Yaskawa INFORM job: DEMO_NAIHAN_0625_2PAINT_0.JBI

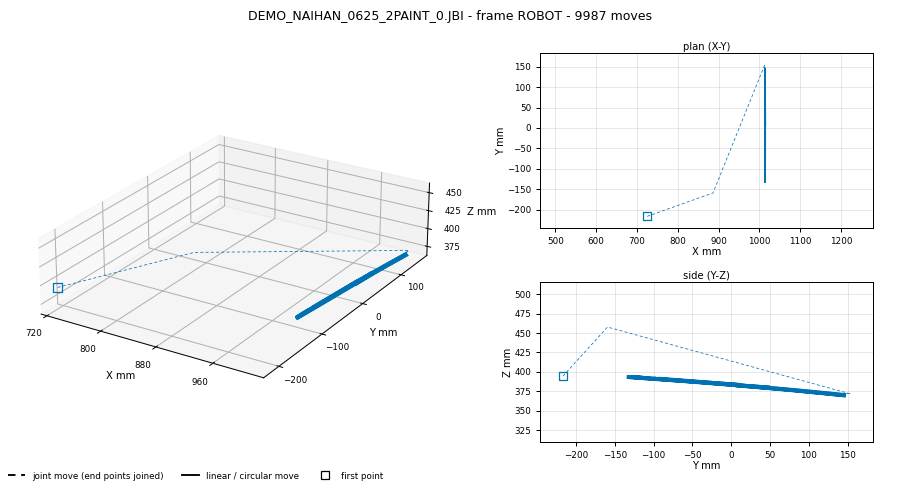
[picture p0: tool path of DEMO_NAIHAN_0625_2PAINT_0.JBI in frame ROBOT, 9987 of 9987 moves have a stored position in this frame; points joined in program order, loops and branches not executed]
/JOB
//NAME DEMO_NAIHAN_0625_2PAINT
//POS
///NPOS 9987,0,0,0,0,0
///TOOL 1
///USER 0
///POSTYPE ROBOT
///RECTAN
///RCONF 1,0,0,0,0,0,0,0,0,0,0,0,0,0,0,0,0,0,0,0,0,0,0,0
C00000=724.889,-216.680,394.500,-180.000,-0.000,-0.000
///USER 0
///POSTYPE ROBOT
///RECTAN
///RCONF 0,0,0,0,0,0,0,0,0,0,0,0,0,0,0,0,0,0,0,0,0,0,0,0
C00001=886.160,-159.406,457.717,-85.028,-4.406,-90.070
///RCONF 1,0,0,0,0,0,0,0,0,0,0,0,0,0,0,0,0,0,0,0,0,0,0,0
C00002=1012.315,153.041,371.808,165.953,61.802,161.272
///RCONF 1,0,0,0,1,0,0,0,0,0,0,0,0,0,0,0,0,0,0,0,0,0,0,0
C00003=1012.444,147.263,372.118,165.953,61.802,161.272
C00004=1012.445,146.855,372.160,165.949,61.816,161.274
C00005=1012.446,146.448,372.202,165.946,61.830,161.276
C00006=1012.447,146.042,372.243,165.944,61.843,161.278
C00007=1012.448,145.637,372.284,165.940,61.857,161.280
C00008=1012.449,145.231,372.325,165.937,61.871,161.282
C00009=1012.450,144.826,372.367,165.934,61.885,161.284
C00010=1012.451,144.422,372.407,165.931,61.898,161.286
C00011=1012.452,144.018,372.449,165.929,61.912,161.288
C00012=1012.453,143.614,372.490,165.925,61.926,161.289
C00013=1012.454,143.211,372.531,165.923,61.939,161.291
C00014=1012.456,142.810,372.572,165.919,61.952,161.293
C00015=1012.456,142.409,372.612,165.917,61.965,161.295
C00016=1012.457,142.007,372.653,165.913,61.979,161.297
C00017=1012.458,141.808,372.673,165.912,61.986,161.298
C00018=1012.459,141.543,372.701,165.910,61.995,161.299
C00019=1012.459,141.136,372.742,165.908,62.008,161.301
C00020=1012.460,140.919,372.763,165.906,62.015,161.302
C00021=1012.461,140.708,372.785,165.904,62.023,161.303
C00022=1012.461,140.481,372.808,165.903,62.030,161.304
C00023=1012.461,140.239,372.832,165.900,62.037,161.305
C00024=1012.462,139.985,372.858,165.899,62.046,161.306
C00025=1012.463,139.724,372.885,165.897,62.054,161.307
C00026=1012.464,139.462,372.911,165.895,62.064,161.309
C00027=1012.464,139.204,372.937,165.894,62.072,161.310
C00028=1012.465,138.956,372.963,165.891,62.080,161.311
C00029=1012.465,138.720,372.986,165.890,62.088,161.312
C00030=1012.466,138.501,373.009,165.889,62.095,161.314
C00031=1012.467,138.104,373.049,165.886,62.107,161.315
C00032=1012.467,137.804,373.079,165.884,62.117,161.316
C00033=1012.469,137.455,373.114,165.882,62.129,161.318
C00034=1012.470,137.112,373.149,165.879,62.140,161.320
C00035=1012.470,136.790,373.181,165.877,62.151,161.321
C00036=1012.471,136.470,373.214,165.875,62.161,161.323
C00037=1012.472,136.129,373.248,165.873,62.172,161.324
C00038=1012.473,135.760,373.285,165.870,62.184,161.326
C00039=1012.474,135.350,373.326,165.867,62.198,161.328
C00040=1012.475,135.091,373.353,165.865,62.207,161.329
C00041=1012.475,134.860,373.376,165.865,62.215,161.331
C00042=1012.476,134.465,373.416,165.862,62.227,161.333
C00043=1012.478,134.070,373.455,165.859,62.240,161.334
C00044=1012.478,133.676,373.495,165.856,62.253,161.336
C00045=1012.479,133.281,373.535,165.854,62.264,161.338
C00046=1012.481,132.887,373.574,165.852,62.276,161.340
C00047=1012.482,132.493,373.615,165.848,62.289,161.341
C00048=1012.482,132.098,373.654,165.846,62.303,161.343
C00049=1012.483,131.704,373.693,165.844,62.316,161.345
C00050=1012.484,131.309,373.733,165.841,62.328,161.347
C00051=1012.486,130.915,373.773,165.839,62.340,161.349
C00052=1012.487,130.520,373.812,165.836,62.353,161.351
C00053=1012.488,130.126,373.852,165.834,62.364,161.352
C00054=1012.489,129.732,373.891,165.831,62.376,161.354
C00055=1012.489,129.338,373.931,165.830,62.388,161.356
C00056=1012.491,128.943,373.970,165.827,62.401,161.358
C00057=1012.492,128.549,374.010,165.824,62.414,161.360
C00058=1012.493,128.154,374.049,165.821,62.426,161.362
C00059=1012.493,127.760,374.089,165.819,62.438,161.363
C00060=1012.495,127.366,374.128,165.816,62.451,161.365
C00061=1012.496,126.972,374.168,165.814,62.463,161.367
C00062=1012.498,126.577,374.207,165.812,62.474,161.368
C00063=1012.498,126.183,374.247,165.810,62.486,161.370
C00064=1012.499,125.789,374.286,165.807,62.498,161.372
C00065=1012.500,125.394,374.325,165.806,62.511,161.374
C00066=1012.501,125.000,374.364,165.803,62.524,161.376
C00067=1012.502,124.605,374.404,165.801,62.535,161.378
C00068=1012.503,124.212,374.444,165.799,62.547,161.380
C00069=1012.504,123.817,374.482,165.796,62.559,161.381
C00070=1012.505,123.422,374.522,165.794,62.571,161.383
C00071=1012.507,123.029,374.561,165.792,62.581,161.385
C00072=1012.507,122.634,374.600,165.790,62.594,161.387
C00073=1012.509,122.240,374.639,165.787,62.606,161.388
C00074=1012.509,121.846,374.679,165.785,62.619,161.391
C00075=1012.511,121.451,374.718,165.783,62.630,161.392
C00076=1012.512,121.057,374.757,165.781,62.642,161.394
C00077=1012.512,120.663,374.797,165.778,62.653,161.395
C00078=1012.514,120.268,374.836,165.776,62.665,161.397
C00079=1012.515,119.874,374.874,165.774,62.675,161.399
C00080=1012.516,119.480,374.914,165.772,62.687,161.401
C00081=1012.517,119.086,374.953,165.769,62.700,161.402
C00082=1012.518,118.692,374.992,165.767,62.712,161.404
C00083=1012.519,118.297,375.031,165.765,62.724,161.406
C00084=1012.520,117.903,375.071,165.764,62.736,161.408
C00085=1012.521,117.509,375.109,165.761,62.747,161.410
C00086=1012.522,117.114,375.149,165.759,62.758,161.411
C00087=1012.524,116.720,375.188,165.757,62.769,161.413
C00088=1012.525,116.326,375.226,165.755,62.780,161.415
C00089=1012.525,115.932,375.266,165.753,62.792,161.417
C00090=1012.526,115.537,375.305,165.750,62.804,161.418
C00091=1012.527,115.143,375.343,165.749,62.816,161.420
C00092=1012.528,114.748,375.383,165.747,62.827,161.422
C00093=1012.529,114.354,375.421,165.745,62.838,161.424
C00094=1012.531,113.960,375.460,165.743,62.849,161.425
C00095=1012.532,113.566,375.499,165.742,62.860,161.427
C00096=1012.532,113.172,375.538,165.739,62.870,161.428
C00097=1012.534,112.777,375.577,165.736,62.882,161.430
C00098=1012.535,112.383,375.616,165.735,62.894,161.432
C00099=1012.536,111.989,375.654,165.732,62.906,161.434
C00100=1012.537,111.594,375.694,165.731,62.917,161.436
C00101=1012.538,111.200,375.732,165.729,62.928,161.437
C00102=1012.539,110.806,375.771,165.726,62.938,161.439
C00103=1012.540,110.412,375.810,165.725,62.949,161.440
C00104=1012.540,110.017,375.849,165.723,62.959,161.442
C00105=1012.542,109.623,375.888,165.722,62.971,161.444
C00106=1012.543,109.229,375.926,165.719,62.982,161.446
C00107=1012.544,108.835,375.965,165.718,62.994,161.448
C00108=1012.545,108.441,376.003,165.715,63.005,161.449
C00109=1012.546,108.045,376.042,165.714,63.016,161.451
C00110=1012.547,107.651,376.081,165.711,63.026,161.452
C00111=1012.548,107.257,376.119,165.710,63.037,161.454
C00112=1012.550,106.863,376.158,165.708,63.047,161.455
C00113=1012.550,106.468,376.197,165.706,63.058,161.457
C00114=1012.551,106.074,376.235,165.704,63.069,161.459
C00115=1012.552,105.680,376.274,165.703,63.080,161.461
C00116=1012.554,105.285,376.313,165.700,63.092,161.463
C00117=1012.555,104.891,376.351,165.698,63.102,161.464
C00118=1012.555,104.496,376.390,165.697,63.113,161.466
C00119=1012.556,104.102,376.428,165.694,63.123,161.467
C00120=1012.557,103.708,376.467,165.693,63.132,161.469
C00121=1012.559,103.314,376.506,165.691,63.142,161.470
C00122=1012.560,102.918,376.544,165.690,63.154,161.472
C00123=1012.561,102.524,376.582,165.688,63.165,161.474
C00124=1012.561,102.130,376.621,165.687,63.176,161.476
C00125=1012.563,101.736,376.659,165.685,63.187,161.478
C00126=1012.563,101.341,376.697,165.683,63.197,161.479
C00127=1012.565,100.946,376.737,165.681,63.207,161.480
C00128=1012.566,100.552,376.774,165.680,63.216,161.482
C00129=1012.567,100.158,376.813,165.678,63.226,161.484
C00130=1012.568,99.764,376.851,165.676,63.237,161.485
C00131=1012.569,99.368,376.889,165.675,63.248,161.487
C00132=1012.569,98.974,376.928,165.673,63.259,161.489
C00133=1012.571,98.580,376.966,165.671,63.269,161.490
C00134=1012.572,98.186,377.004,165.669,63.279,161.492
C00135=1012.573,97.790,377.043,165.667,63.289,161.493
C00136=1012.574,97.396,377.081,165.665,63.298,161.495
C00137=1012.575,97.001,377.119,165.664,63.308,161.496
C00138=1012.576,96.607,377.158,165.662,63.318,161.498
C00139=1012.577,96.212,377.196,165.661,63.329,161.500
C00140=1012.578,95.818,377.234,165.659,63.340,161.502
C00141=1012.579,95.423,377.272,165.657,63.350,161.503
C00142=1012.580,95.029,377.310,165.655,63.360,161.504
C00143=1012.581,94.634,377.349,165.654,63.369,161.506
C00144=1012.582,94.239,377.386,165.652,63.380,161.507
C00145=1012.583,93.845,377.425,165.650,63.388,161.509
C00146=1012.583,93.450,377.463,165.649,63.398,161.510
C00147=1012.585,93.055,377.501,165.648,63.407,161.512
C00148=1012.586,92.660,377.539,165.646,63.418,161.513
C00149=1012.586,92.266,377.577,165.643,63.428,161.515
C00150=1012.588,91.871,377.615,165.643,63.438,161.517
C00151=1012.589,91.476,377.653,165.641,63.448,161.518
C00152=1012.590,91.074,377.692,165.639,63.458,161.520
C00153=1012.590,90.827,377.715,165.639,63.464,161.521
C00154=1012.590,90.548,377.743,165.637,63.470,161.522
C00155=1012.592,90.273,377.769,165.636,63.476,161.523
C00156=1012.592,90.039,377.792,165.635,63.482,161.523
C00157=1012.594,89.643,377.830,165.634,63.491,161.525
C00158=1012.595,89.258,377.867,165.632,63.501,161.527
C00159=1012.596,88.879,377.903,165.630,63.510,161.528
C00160=1012.596,88.505,377.940,165.630,63.519,161.530
C00161=1012.598,88.127,377.975,165.628,63.528,161.531
C00162=1012.598,87.742,378.012,165.625,63.537,161.532
C00163=1012.599,87.348,378.050,165.624,63.547,161.534
C00164=1012.600,86.949,378.088,165.623,63.556,161.535
C00165=1012.601,86.548,378.127,165.622,63.566,161.537
C00166=1012.602,86.146,378.166,165.619,63.575,161.538
C00167=1012.603,85.742,378.204,165.618,63.585,161.540
C00168=1012.604,85.338,378.243,165.617,63.595,161.541
C00169=1012.605,84.933,378.282,165.615,63.605,161.543
C00170=1012.605,84.526,378.321,165.613,63.613,161.544
C00171=1012.607,84.117,378.359,165.612,63.623,161.546
C00172=1012.608,83.707,378.399,165.610,63.633,161.547
C00173=1012.608,83.297,378.438,165.609,63.643,161.549
C00174=1012.610,82.884,378.478,165.608,63.652,161.551
C00175=1012.610,82.472,378.517,165.605,63.662,161.552
C00176=1012.612,82.058,378.556,165.604,63.671,161.553
C00177=1012.613,81.643,378.596,165.603,63.681,161.555
C00178=1012.614,81.249,378.633,165.601,63.690,161.556
C00179=1012.614,80.886,378.668,165.599,63.699,161.558
C00180=1012.616,80.503,378.704,165.599,63.707,161.559
C00181=1012.616,80.090,378.744,165.597,63.716,161.560
C00182=1012.617,79.682,378.782,165.595,63.726,161.562
C00183=1012.618,79.279,378.821,165.594,63.734,161.563
C00184=1012.619,78.885,378.858,165.592,63.743,161.565
C00185=1012.620,78.495,378.896,165.590,63.752,161.566
C00186=1012.621,78.112,378.932,165.589,63.761,161.567
C00187=1012.622,77.730,378.968,165.588,63.769,161.569
C00188=1012.623,77.348,379.004,165.586,63.778,161.570
C00189=1012.623,76.961,379.041,165.585,63.786,161.571
C00190=1012.624,76.567,379.078,165.584,63.795,161.573
C00191=1012.626,76.165,379.116,165.582,63.804,161.574
C00192=1012.626,75.757,379.155,165.580,63.813,161.575
C00193=1012.627,75.342,379.194,165.579,63.823,161.577
C00194=1012.627,75.133,379.214,165.578,63.826,161.578
C00195=1012.628,74.918,379.234,165.577,63.831,161.578
C00196=1012.628,74.691,379.256,165.576,63.836,161.579
C00197=1012.629,74.463,379.277,165.576,63.841,161.580
C00198=1012.629,74.244,379.297,165.575,63.846,161.581
C00199=1012.631,73.829,379.338,165.574,63.855,161.582
C00200=1012.631,73.417,379.376,165.572,63.864,161.583
C00201=1012.632,73.008,379.414,165.570,63.873,161.585
C00202=1012.633,72.599,379.453,165.569,63.881,161.586
C00203=1012.633,72.194,379.492,165.568,63.890,161.587
C00204=1012.635,71.788,379.530,165.566,63.899,161.589
C00205=1012.636,71.383,379.568,165.565,63.907,161.590
C00206=1012.637,70.980,379.606,165.563,63.916,161.592
C00207=1012.637,70.574,379.644,165.562,63.925,161.593
C00208=1012.638,70.170,379.682,165.561,63.933,161.594
C00209=1012.640,69.766,379.720,165.559,63.942,161.596
C00210=1012.640,69.358,379.758,165.558,63.950,161.597
C00211=1012.641,68.942,379.797,165.556,63.959,161.598
C00212=1012.641,68.523,379.836,165.554,63.967,161.599
C00213=1012.643,68.112,379.875,165.553,63.976,161.601
C00214=1012.643,67.711,379.912,165.552,63.985,161.602
C00215=1012.645,67.313,379.950,165.550,63.992,161.603
C00216=1012.645,66.915,379.987,165.550,64.001,161.605
C00217=1012.646,66.551,380.022,165.548,64.008,161.606
C00218=1012.647,66.224,380.052,165.547,64.015,161.607
C00219=1012.647,65.831,380.088,165.545,64.022,161.608
C00220=1012.648,65.623,380.108,165.545,64.027,161.609
C00221=1012.648,65.408,380.128,165.544,64.031,161.609
C00222=1012.649,65.189,380.149,165.544,64.036,161.610
C00223=1012.649,64.966,380.169,165.542,64.040,161.611
C00224=1012.649,64.740,380.191,165.542,64.045,161.612
C00225=1012.651,64.514,380.212,165.540,64.049,161.612
C00226=1012.651,64.295,380.232,165.540,64.053,161.613
C00227=1012.651,63.890,380.269,165.537,64.085,161.619
C00228=1012.650,63.679,380.286,165.536,64.150,161.632
C00229=1012.649,63.443,380.305,165.533,64.223,161.647
C00230=1012.648,63.194,380.324,165.530,64.299,161.663
C00231=1012.647,62.952,380.344,165.527,64.374,161.678
C00232=1012.646,62.733,380.362,165.524,64.440,161.692
C00233=1012.645,62.450,380.384,165.522,64.527,161.710
C00234=1012.644,62.051,380.416,165.518,64.647,161.735
C00235=1012.641,61.654,380.447,165.515,64.765,161.760
C00236=1012.640,61.259,380.479,165.512,64.884,161.785
C00237=1012.639,60.863,380.511,165.509,65.001,161.810
C00238=1012.637,60.466,380.543,165.507,65.118,161.835
C00239=1012.635,60.071,380.574,165.504,65.234,161.859
C00240=1012.634,59.675,380.606,165.502,65.350,161.884
C00241=1012.633,59.278,380.638,165.501,65.464,161.910
C00242=1012.631,58.883,380.669,165.499,65.578,161.934
C00243=1012.630,58.486,380.701,165.498,65.692,161.960
C00244=1012.629,58.090,380.733,165.496,65.805,161.985
C00245=1012.627,57.695,380.765,165.496,65.917,162.010
C00246=1012.626,57.298,380.797,165.495,66.028,162.035
C00247=1012.625,56.902,380.828,165.496,66.139,162.060
C00248=1012.624,56.507,380.860,165.496,66.249,162.085
C00249=1012.623,56.110,380.892,165.496,66.358,162.110
C00250=1012.621,55.714,380.924,165.496,66.467,162.135
C00251=1012.620,55.318,380.955,165.496,66.576,162.160
C00252=1012.619,54.922,380.987,165.497,66.683,162.185
C00253=1012.617,54.527,381.019,165.499,66.791,162.211
C00254=1012.616,54.130,381.051,165.500,66.896,162.235
C00255=1012.615,53.734,381.083,165.501,67.002,162.261
C00256=1012.614,53.339,381.115,165.503,67.108,162.286
C00257=1012.613,52.942,381.146,165.506,67.213,162.311
C00258=1012.611,52.547,381.178,165.508,67.317,162.337
C00259=1012.611,52.151,381.210,165.510,67.419,162.362
C00260=1012.609,51.754,381.242,165.513,67.522,162.387
C00261=1012.608,51.358,381.274,165.516,67.624,162.412
C00262=1012.607,50.963,381.306,165.520,67.726,162.438
C00263=1012.606,50.567,381.338,165.523,67.827,162.463
C00264=1012.605,50.171,381.369,165.528,67.928,162.489
C00265=1012.604,49.775,381.401,165.530,68.028,162.514
C00266=1012.603,49.380,381.433,165.536,68.127,162.540
C00267=1012.602,48.983,381.465,165.539,68.226,162.565
C00268=1012.601,48.588,381.496,165.543,68.324,162.591
C00269=1012.600,48.192,381.528,165.550,68.421,162.617
C00270=1012.599,47.796,381.561,165.554,68.518,162.642
C00271=1012.598,47.400,381.592,165.560,68.615,162.668
C00272=1012.597,47.005,381.624,165.564,68.710,162.693
C00273=1012.597,46.610,381.656,165.571,68.806,162.719
C00274=1012.596,46.214,381.688,165.576,68.901,162.745
C00275=1012.595,45.818,381.719,165.582,68.994,162.771
C00276=1012.594,45.422,381.751,165.588,69.088,162.796
C00277=1012.593,45.026,381.783,165.594,69.181,162.822
C00278=1012.592,44.630,381.816,165.602,69.274,162.848
C00279=1012.592,44.236,381.847,165.608,69.365,162.874
C00280=1012.591,43.839,381.879,165.616,69.457,162.900
C00281=1012.590,43.443,381.911,165.623,69.547,162.926
C00282=1012.589,43.048,381.943,165.630,69.637,162.952
C00283=1012.588,42.653,381.975,165.639,69.727,162.978
C00284=1012.588,42.257,382.007,165.646,69.816,163.004
C00285=1012.587,41.861,382.038,165.655,69.905,163.030
C00286=1012.586,41.466,382.070,165.663,69.993,163.056
C00287=1012.586,41.070,382.103,165.671,70.080,163.082
C00288=1012.585,40.675,382.134,165.680,70.167,163.108
C00289=1012.584,40.280,382.166,165.689,70.253,163.134
C00290=1012.584,39.884,382.199,165.698,70.338,163.160
C00291=1012.583,39.489,382.230,165.708,70.424,163.187
C00292=1012.582,39.093,382.261,165.716,70.508,163.213
C00293=1012.582,38.697,382.294,165.727,70.592,163.240
C00294=1012.581,38.302,382.325,165.737,70.676,163.266
C00295=1012.581,37.906,382.358,165.747,70.758,163.292
C00296=1012.580,37.511,382.390,165.756,70.841,163.318
C00297=1012.579,37.116,382.421,165.767,70.922,163.345
C00298=1012.579,36.720,382.454,165.778,71.004,163.371
C00299=1012.578,36.325,382.486,165.788,71.084,163.397
C00300=1012.578,35.930,382.518,165.799,71.164,163.424
C00301=1012.576,35.534,382.550,165.810,71.243,163.450
C00302=1012.576,35.139,382.581,165.820,71.322,163.476
C00303=1012.576,34.744,382.613,165.832,71.401,163.503
C00304=1012.575,34.348,382.645,165.843,71.478,163.529
C00305=1012.575,33.953,382.677,165.855,71.556,163.556
C00306=1012.574,33.557,382.709,165.867,71.631,163.581
C00307=1012.574,33.162,382.741,165.878,71.707,163.608
C00308=1012.573,32.767,382.772,165.891,71.782,163.634
C00309=1012.573,32.371,382.805,165.903,71.857,163.661
C00310=1012.572,31.976,382.837,165.916,71.931,163.687
C00311=1012.572,31.580,382.869,165.928,72.005,163.713
C00312=1012.571,31.185,382.901,165.940,72.077,163.739
C00313=1012.571,30.790,382.933,165.953,72.149,163.765
C00314=1012.571,30.395,382.964,165.966,72.221,163.792
C00315=1012.570,29.999,382.997,165.978,72.292,163.818
C00316=1012.570,29.604,383.029,165.990,72.362,163.843
C00317=1012.570,29.209,383.061,166.004,72.432,163.870
C00318=1012.569,28.815,383.093,166.017,72.502,163.896
C00319=1012.568,28.420,383.125,166.030,72.569,163.921
C00320=1012.568,28.028,383.157,166.043,72.636,163.947
C00321=1012.568,27.634,383.189,166.058,72.703,163.973
C00322=1012.568,27.241,383.221,166.071,72.769,163.998
C00323=1012.567,26.847,383.253,166.085,72.835,164.024
C00324=1012.566,26.450,383.285,166.097,72.900,164.049
C00325=1012.566,26.053,383.318,166.111,72.965,164.075
C00326=1012.566,25.645,383.350,166.124,73.031,164.100
C00327=1012.608,25.661,383.471,165.674,70.447,163.177
C00328=1012.650,25.676,383.593,165.454,67.873,162.444
C00329=1012.652,26.075,383.563,165.449,67.750,162.412
C00330=1012.653,26.473,383.533,165.445,67.626,162.382
C00331=1012.656,26.869,383.504,165.440,67.503,162.350
C00332=1012.657,27.264,383.475,165.437,67.380,162.320
C00333=1012.659,27.657,383.446,165.433,67.258,162.290
C00334=1012.660,28.050,383.416,165.431,67.135,162.261
C00335=1012.662,28.443,383.386,165.427,67.013,162.231
C00336=1012.664,28.838,383.357,165.425,66.890,162.202
C00337=1012.666,29.233,383.327,165.423,66.766,162.173
C00338=1012.667,29.629,383.298,165.422,66.642,162.144
C00339=1012.669,30.024,383.268,165.421,66.519,162.115
C00340=1012.671,30.420,383.239,165.420,66.395,162.087
C00341=1012.673,30.815,383.210,165.418,66.270,162.058
C00342=1012.675,31.211,383.179,165.419,66.146,162.030
C00343=1012.676,31.606,383.150,165.419,66.022,162.002
C00344=1012.679,32.002,383.120,165.419,65.898,161.974
C00345=1012.680,32.397,383.091,165.420,65.772,161.946
C00346=1012.683,32.793,383.061,165.420,65.648,161.918
C00347=1012.684,33.188,383.031,165.422,65.523,161.891
C00348=1012.686,33.584,383.001,165.423,65.398,161.864
C00349=1012.688,33.980,382.971,165.425,65.272,161.837
C00350=1012.690,34.375,382.942,165.427,65.148,161.810
C00351=1012.692,34.770,382.912,165.430,65.022,161.783
C00352=1012.694,35.167,382.882,165.433,64.896,161.756
C00353=1012.695,35.562,382.852,165.436,64.771,161.730
C00354=1012.698,35.957,382.822,165.439,64.645,161.704
C00355=1012.700,36.353,382.792,165.442,64.520,161.677
C00356=1012.701,36.748,382.762,165.446,64.393,161.651
C00357=1012.703,37.144,382.732,165.450,64.267,161.625
C00358=1012.706,37.540,382.702,165.454,64.141,161.599
C00359=1012.707,37.936,382.672,165.459,64.015,161.574
C00360=1012.710,38.331,382.642,165.465,63.888,161.549
C00361=1012.711,38.726,382.612,165.469,63.762,161.523
C00362=1012.713,39.122,382.581,165.475,63.635,161.498
C00363=1012.716,39.518,382.551,165.481,63.509,161.473
C00364=1012.718,39.913,382.521,165.486,63.382,161.448
C00365=1012.720,40.309,382.491,165.493,63.255,161.423
C00366=1012.722,40.705,382.461,165.500,63.128,161.398
C00367=1012.724,41.100,382.431,165.506,63.002,161.373
C00368=1012.726,41.496,382.400,165.513,62.874,161.349
C00369=1012.728,41.892,382.370,165.520,62.747,161.324
C00370=1012.731,42.287,382.340,165.528,62.620,161.300
C00371=1012.732,42.683,382.309,165.535,62.493,161.276
C00372=1012.735,43.079,382.279,165.544,62.367,161.252
C00373=1012.736,43.475,382.249,165.552,62.238,161.228
C00374=1012.739,43.871,382.218,165.561,62.112,161.204
C00375=1012.741,44.267,382.188,165.569,61.985,161.180
C00376=1012.743,44.662,382.158,165.577,61.857,161.156
C00377=1012.745,45.058,382.127,165.587,61.730,161.133
C00378=1012.748,45.454,382.097,165.596,61.602,161.110
C00379=1012.750,45.850,382.066,165.606,61.475,161.086
C00380=1012.752,46.245,382.035,165.615,61.347,161.063
C00381=1012.754,46.641,382.005,165.626,61.220,161.040
C00382=1012.757,47.038,381.974,165.636,61.092,161.017
C00383=1012.759,47.434,381.944,165.646,60.965,160.994
C00384=1012.761,47.829,381.914,165.657,60.838,160.971
C00385=1012.764,48.225,381.882,165.668,60.711,160.948
C00386=1012.765,48.621,381.851,165.678,60.584,160.925
C00387=1012.768,49.017,381.821,165.691,60.456,160.903
C00388=1012.770,49.413,381.789,165.702,60.329,160.881
C00389=1012.773,49.809,381.759,165.714,60.202,160.858
C00390=1012.773,49.925,381.750,165.718,60.165,160.852
C00391=1012.563,19.548,383.847,166.338,73.918,164.472
C00392=1012.562,19.333,383.865,166.346,73.946,164.485
C00393=1012.562,18.920,383.898,166.359,73.998,164.508
C00394=1012.563,18.696,383.916,166.367,74.026,164.520
C00395=1012.562,18.447,383.937,166.375,74.057,164.534
C00396=1012.562,18.198,383.957,166.384,74.088,164.548
C00397=1012.562,17.950,383.977,166.391,74.118,164.561
C00398=1012.562,17.704,383.997,166.400,74.147,164.575
C00399=1012.562,17.454,384.018,166.408,74.177,164.588
C00400=1012.562,17.207,384.038,166.416,74.205,164.601
C00401=1012.562,16.960,384.058,166.423,74.233,164.613
C00402=1012.562,16.714,384.079,166.432,74.261,164.626
C00403=1012.562,16.464,384.099,166.439,74.288,164.639
C00404=1012.561,16.216,384.119,166.446,74.315,164.651
C00405=1012.561,15.968,384.139,166.455,74.342,164.663
C00406=1012.562,15.722,384.161,166.463,74.368,164.676
C00407=1012.562,15.472,384.181,166.470,74.394,164.688
C00408=1012.561,15.223,384.202,166.477,74.419,164.699
C00409=1012.562,14.975,384.222,166.484,74.444,164.710
C00410=1012.562,14.726,384.243,166.491,74.467,164.722
C00411=1012.562,14.476,384.263,166.496,74.491,164.732
C00412=1012.562,14.227,384.283,166.504,74.514,164.744
C00413=1012.561,13.977,384.304,166.512,74.537,164.755
C00414=1012.561,13.727,384.325,166.518,74.558,164.764
C00415=1012.561,13.478,384.345,166.524,74.580,164.774
C00416=1012.562,13.227,384.366,166.529,74.600,164.784
C00417=1012.562,12.977,384.387,166.536,74.619,164.793
C00418=1012.562,12.727,384.408,166.541,74.640,164.803
C00419=1012.562,12.478,384.429,166.546,74.657,164.810
C00420=1012.562,12.230,384.449,166.551,74.674,164.818
C00421=1012.562,11.984,384.470,166.556,74.691,164.827
C00422=1012.562,11.745,384.490,166.560,74.706,164.833
C00423=1012.562,11.497,384.511,166.566,74.721,164.841
C00424=1012.562,11.251,384.532,166.569,74.734,164.847
C00425=1012.563,11.001,384.552,166.573,74.747,164.853
C00426=1012.562,10.747,384.574,166.576,74.758,164.859
C00427=1012.563,10.497,384.595,166.578,74.769,164.863
C00428=1012.562,10.247,384.616,166.581,74.777,164.867
C00429=1012.563,9.999,384.637,166.584,74.784,164.871
C00430=1012.563,9.750,384.659,166.583,74.790,164.872
C00431=1012.564,9.502,384.680,166.585,74.793,164.875
C00432=1012.564,9.253,384.701,166.584,74.794,164.874
C00433=1012.564,9.005,384.723,166.584,74.792,164.873
C00434=1012.564,8.756,384.744,166.581,74.789,164.871
C00435=1012.564,8.508,384.766,166.578,74.780,164.866
C00436=1012.565,8.257,384.789,166.573,74.768,164.860
C00437=1012.566,8.007,384.811,166.565,74.749,164.849
C00438=1012.566,7.756,384.834,166.555,74.723,164.836
C00439=1012.567,7.505,384.857,166.543,74.684,164.817
C00440=1012.569,7.092,384.899,166.501,74.562,164.756
C00441=1012.572,6.931,384.924,166.429,74.336,164.647
C00442=1012.576,7.213,384.915,166.334,74.017,164.499
C00443=1012.579,7.492,384.899,166.286,73.844,164.421
C00444=1012.579,7.769,384.882,166.248,73.701,164.359
C00445=1012.581,8.044,384.864,166.213,73.571,164.302
C00446=1012.582,8.293,384.849,166.187,73.462,164.256
C00447=1012.584,8.542,384.832,166.159,73.358,164.212
C00448=1012.585,8.790,384.815,166.135,73.258,164.170
C00449=1012.586,9.037,384.799,166.113,73.162,164.131
C00450=1012.587,9.286,384.782,166.092,73.068,164.093
C00451=1012.588,9.536,384.765,166.070,72.975,164.055
C00452=1012.589,9.786,384.747,166.050,72.884,164.019
C00453=1012.591,10.036,384.730,166.032,72.794,163.984
C00454=1012.591,10.286,384.712,166.011,72.706,163.948
C00455=1012.592,10.537,384.695,165.994,72.620,163.916
C00456=1012.593,10.787,384.677,165.976,72.534,163.882
C00457=1012.594,11.035,384.661,165.960,72.449,163.850
C00458=1012.595,11.282,384.643,165.943,72.366,163.819
C00459=1012.596,11.527,384.625,165.928,72.284,163.789
C00460=1012.597,11.773,384.608,165.911,72.202,163.758
C00461=1012.598,12.024,384.590,165.897,72.120,163.728
C00462=1012.599,12.276,384.572,165.882,72.037,163.698
C00463=1012.599,12.531,384.554,165.867,71.954,163.667
C00464=1012.600,12.787,384.535,165.852,71.872,163.638
C00465=1012.602,13.042,384.518,165.839,71.789,163.609
C00466=1012.602,13.291,384.500,165.825,71.709,163.581
C00467=1012.603,13.540,384.482,165.812,71.630,163.553
C00468=1012.604,13.788,384.464,165.801,71.552,163.526
C00469=1012.605,14.037,384.446,165.788,71.472,163.499
C00470=1012.606,14.286,384.428,165.775,71.394,163.472
C00471=1012.607,14.535,384.410,165.765,71.316,163.446
C00472=1012.608,14.784,384.392,165.752,71.237,163.419
C00473=1012.609,15.032,384.375,165.742,71.159,163.393
C00474=1012.609,15.281,384.357,165.731,71.082,163.368
C00475=1012.611,15.530,384.338,165.720,71.003,163.342
C00476=1012.611,15.780,384.320,165.709,70.926,163.317
C00477=1012.612,16.030,384.302,165.698,70.848,163.291
C00478=1012.613,16.279,384.283,165.689,70.771,163.267
C00479=1012.614,16.530,384.266,165.679,70.693,163.242
C00480=1012.616,16.780,384.247,165.670,70.616,163.217
C00481=1012.616,17.032,384.229,165.660,70.538,163.193
C00482=1012.617,17.282,384.211,165.650,70.460,163.168
C00483=1012.618,17.532,384.193,165.643,70.383,163.145
C00484=1012.619,17.784,384.174,165.634,70.305,163.121
C00485=1012.620,18.035,384.157,165.625,70.228,163.097
C00486=1012.621,18.285,384.138,165.616,70.151,163.073
C00487=1012.622,18.536,384.119,165.608,70.074,163.050
C00488=1012.623,18.787,384.101,165.602,69.997,163.027
C00489=1012.624,19.039,384.083,165.593,69.919,163.004
C00490=1012.625,19.445,384.053,165.582,69.794,162.967
C00491=1012.627,19.860,384.022,165.570,69.666,162.930
C00492=1012.628,20.097,384.005,165.563,69.594,162.909
C00493=1012.629,20.355,383.986,165.556,69.515,162.886
C00494=1012.630,20.622,383.966,165.548,69.432,162.862
C00495=1012.631,20.890,383.947,165.543,69.350,162.839
C00496=1012.632,21.151,383.928,165.536,69.270,162.816
C00497=1012.633,21.394,383.910,165.530,69.195,162.795
C00498=1012.634,21.619,383.893,165.525,69.125,162.776
C00499=1012.636,22.009,383.864,165.516,69.005,162.742
C00500=1012.637,22.235,383.847,165.511,68.936,162.723
C00501=1012.637,22.496,383.828,165.505,68.855,162.701
C00502=1012.638,22.731,383.811,165.502,68.783,162.682
C00503=1012.639,22.936,383.796,165.498,68.720,162.665
C00504=1012.640,23.172,383.778,165.492,68.647,162.645
C00505=1012.641,23.403,383.762,165.488,68.576,162.626
C00506=1012.642,23.662,383.742,165.485,68.496,162.605
C00507=1012.643,23.967,383.719,165.479,68.402,162.580
C00508=1012.645,24.277,383.697,165.474,68.306,162.555
C00509=1012.645,24.606,383.672,165.468,68.204,162.528
C00510=1012.647,24.943,383.647,165.463,68.100,162.501
C00511=1012.649,25.279,383.622,165.459,67.996,162.475
C00512=1012.608,25.267,383.502,165.684,70.540,163.205
C00513=1012.566,25.254,383.382,166.140,73.093,164.126
C00514=1012.566,25.655,383.349,166.125,73.029,164.100
C00515=1012.566,25.407,383.369,166.134,73.069,164.116
C00516=1012.566,25.161,383.389,166.142,73.108,164.131
C00517=1012.565,24.749,383.423,166.157,73.173,164.158
C00518=1012.606,24.817,383.537,165.697,70.641,163.237
C00519=1012.566,24.864,383.414,166.152,73.155,164.150
C00520=1012.567,25.258,383.381,166.139,73.092,164.126
C00521=1012.566,25.009,383.401,166.147,73.131,164.141
C00522=1012.565,24.758,383.422,166.156,73.171,164.157
C00523=1012.566,24.509,383.442,166.165,73.210,164.173
C00524=1012.566,24.265,383.462,166.174,73.247,164.188
C00525=1012.565,24.022,383.482,166.183,73.284,164.204
C00526=1012.565,23.799,383.500,166.190,73.318,164.217
C00527=1012.565,23.420,383.531,166.204,73.376,164.242
C00528=1012.565,23.183,383.550,166.211,73.411,164.256
C00529=1012.564,22.945,383.569,166.220,73.446,164.270
C00530=1012.564,22.675,383.592,166.229,73.487,164.287
C00531=1012.564,22.351,383.618,166.241,73.534,164.307
C00532=1012.564,22.116,383.637,166.249,73.567,164.321
C00533=1012.564,21.885,383.656,166.257,73.601,164.335
C00534=1012.564,21.597,383.679,166.268,73.641,164.353
C00535=1012.563,21.269,383.706,166.279,73.687,164.372
C00536=1012.563,21.013,383.727,166.287,73.722,164.387
C00537=1012.563,20.748,383.749,166.297,73.758,164.403
C00538=1012.564,20.478,383.770,166.306,73.795,164.419
C00539=1012.563,20.214,383.792,166.316,73.831,164.435
C00540=1012.563,19.973,383.812,166.323,73.862,164.448
C00541=1012.563,19.751,383.830,166.330,73.892,164.461
C00542=1012.563,19.548,383.847,166.338,73.918,164.472
C00543=1012.629,-93.771,392.738,165.388,72.408,163.533
C00544=1012.625,-93.572,392.712,165.447,72.663,163.632
C00545=1012.618,-93.811,392.708,165.547,73.088,163.799
C00546=1012.618,-94.073,392.721,165.566,73.174,163.833
C00547=1012.616,-94.335,392.737,165.578,73.226,163.853
C00548=1012.616,-94.597,392.752,165.586,73.262,163.867
C00549=1012.640,-94.959,392.854,165.225,71.642,163.251
C00550=1012.643,-95.343,392.888,165.187,71.445,163.182
C00551=1012.645,-95.723,392.922,165.153,71.261,163.119
C00552=1012.648,-96.102,392.956,165.121,71.084,163.059
C00553=1012.615,-96.298,392.863,165.586,73.314,163.882
C00554=1012.651,-96.479,392.988,165.090,70.913,163.001
C00555=1012.649,-96.226,392.966,165.112,71.028,163.040
C00556=1012.647,-95.971,392.944,165.130,71.144,163.078
C00557=1012.646,-95.723,392.922,165.154,71.262,163.120
C00558=1012.643,-95.472,392.900,165.176,71.382,163.161
C00559=1012.642,-95.223,392.877,165.200,71.506,163.204
C00560=1012.641,-94.972,392.854,165.224,71.635,163.249
C00561=1012.638,-94.723,392.832,165.251,71.769,163.297
C00562=1012.636,-94.473,392.809,165.281,71.911,163.349
C00563=1012.634,-94.223,392.784,165.314,72.066,163.406
C00564=1012.631,-93.972,392.759,165.351,72.240,163.470
C00565=1012.629,-93.771,392.738,165.388,72.408,163.533
C00566=1012.844,-122.010,395.059,164.569,61.082,160.666
C00567=1012.842,-121.711,395.036,164.565,61.193,160.686
C00568=1012.838,-121.322,395.007,164.561,61.338,160.712
C00569=1012.835,-120.934,394.976,164.556,61.483,160.738
C00570=1012.831,-120.546,394.946,164.553,61.628,160.765
C00571=1012.828,-120.157,394.916,164.549,61.773,160.792
C00572=1012.824,-119.769,394.885,164.546,61.919,160.819
C00573=1012.821,-119.380,394.855,164.542,62.064,160.845
C00574=1012.817,-118.992,394.825,164.541,62.210,160.873
C00575=1012.814,-118.604,394.794,164.538,62.356,160.900
C00576=1012.811,-118.215,394.764,164.536,62.502,160.928
C00577=1012.808,-117.827,394.734,164.534,62.647,160.956
C00578=1012.805,-117.439,394.703,164.532,62.794,160.984
C00579=1012.801,-117.050,394.672,164.532,62.940,161.012
C00580=1012.798,-116.661,394.642,164.531,63.087,161.041
C00581=1012.795,-116.273,394.612,164.530,63.233,161.069
C00582=1012.791,-115.885,394.580,164.530,63.379,161.098
C00583=1012.788,-115.496,394.550,164.530,63.526,161.127
C00584=1012.785,-115.107,394.519,164.530,63.673,161.157
C00585=1012.782,-114.718,394.488,164.531,63.819,161.186
C00586=1012.779,-114.330,394.457,164.532,63.966,161.216
C00587=1012.776,-113.942,394.426,164.533,64.114,161.246
C00588=1012.772,-113.553,394.395,164.535,64.260,161.276
C00589=1012.770,-113.164,394.364,164.538,64.407,161.307
C00590=1012.767,-112.775,394.333,164.540,64.554,161.338
C00591=1012.764,-112.387,394.302,164.542,64.701,161.369
C00592=1012.760,-111.998,394.271,164.546,64.848,161.400
C00593=1012.757,-111.610,394.240,164.550,64.995,161.432
C00594=1012.755,-111.221,394.208,164.554,65.143,161.464
C00595=1012.752,-110.832,394.178,164.558,65.290,161.496
C00596=1012.749,-110.443,394.146,164.564,65.437,161.528
C00597=1012.746,-110.054,394.115,164.568,65.584,161.561
C00598=1012.743,-109.665,394.083,164.574,65.732,161.594
C00599=1012.740,-109.276,394.052,164.581,65.880,161.627
C00600=1012.737,-108.871,394.019,164.587,66.033,161.662
C00601=1012.735,-108.660,394.001,164.591,66.113,161.681
C00602=1012.734,-108.441,393.985,164.595,66.196,161.700
C00603=1012.732,-108.216,393.966,164.599,66.282,161.720
C00604=1012.731,-107.987,393.947,164.604,66.369,161.740
C00605=1012.729,-107.754,393.929,164.607,66.457,161.760
C00606=1012.727,-107.521,393.910,164.612,66.545,161.781
C00607=1012.725,-107.292,393.891,164.616,66.633,161.802
C00608=1012.723,-107.065,393.872,164.622,66.719,161.822
C00609=1012.722,-106.844,393.855,164.626,66.803,161.843
C00610=1012.719,-106.424,393.820,164.637,66.963,161.881
C00611=1012.717,-106.027,393.788,164.646,67.114,161.918
C00612=1012.714,-105.638,393.756,164.658,67.262,161.955
C00613=1012.671,-105.646,393.637,164.865,69.785,162.620
C00614=1012.629,-105.653,393.519,165.277,72.316,163.451
C00615=1012.630,-106.043,393.547,165.262,72.255,163.427
C00616=1012.631,-106.440,393.575,165.246,72.191,163.402
C00617=1012.632,-106.860,393.606,165.228,72.121,163.374
C00618=1012.633,-107.082,393.622,165.219,72.084,163.360
C00619=1012.633,-107.307,393.638,165.209,72.045,163.345
C00620=1012.633,-107.537,393.654,165.198,72.006,163.330
C00621=1012.634,-107.770,393.671,165.190,71.967,163.315
C00622=1012.635,-108.002,393.688,165.181,71.926,163.300
C00623=1012.636,-108.232,393.704,165.171,71.886,163.285
C00624=1012.637,-108.457,393.720,165.161,71.846,163.269
C00625=1012.637,-108.677,393.736,165.152,71.807,163.255
C00626=1012.638,-109.094,393.766,165.134,71.732,163.227
C00627=1012.639,-109.489,393.795,165.117,71.660,163.200
C00628=1012.640,-109.877,393.822,165.101,71.587,163.173
C00629=1012.641,-110.266,393.851,165.084,71.514,163.146
C00630=1012.643,-110.656,393.879,165.069,71.440,163.120
C00631=1012.643,-111.045,393.907,165.053,71.365,163.093
C00632=1012.644,-111.433,393.935,165.036,71.289,163.066
C00633=1012.646,-111.822,393.964,165.020,71.212,163.039
C00634=1012.647,-112.211,393.991,165.004,71.134,163.011
C00635=1012.648,-112.600,394.019,164.987,71.054,162.983
C00636=1012.649,-112.989,394.048,164.972,70.975,162.956
C00637=1012.651,-113.378,394.075,164.957,70.894,162.929
C00638=1012.652,-113.767,394.103,164.941,70.812,162.901
C00639=1012.653,-114.155,394.131,164.925,70.729,162.873
C00640=1012.655,-114.544,394.160,164.908,70.645,162.845
C00641=1012.656,-114.933,394.188,164.893,70.561,162.817
C00642=1012.657,-115.321,394.217,164.879,70.475,162.790
C00643=1012.659,-115.710,394.244,164.864,70.389,162.762
C00644=1012.661,-116.099,394.273,164.849,70.301,162.733
C00645=1012.662,-116.487,394.300,164.833,70.213,162.705
C00646=1012.663,-116.876,394.329,164.819,70.124,162.677
C00647=1012.664,-117.264,394.357,164.804,70.035,162.649
C00648=1012.666,-117.653,394.385,164.789,69.944,162.620
C00649=1012.668,-118.041,394.414,164.775,69.852,162.592
C00650=1012.669,-118.430,394.442,164.761,69.759,162.563
C00651=1012.671,-118.818,394.470,164.746,69.665,162.535
C00652=1012.673,-119.207,394.499,164.733,69.570,162.506
C00653=1012.674,-119.595,394.527,164.719,69.475,162.478
C00654=1012.675,-119.984,394.555,164.707,69.379,162.450
C00655=1012.677,-120.372,394.584,164.693,69.281,162.421
C00656=1012.678,-120.761,394.612,164.680,69.183,162.393
C00657=1012.680,-121.149,394.640,164.667,69.083,162.364
C00658=1012.682,-121.537,394.669,164.654,68.983,162.335
C00659=1012.684,-121.926,394.697,164.641,68.882,162.306
C00660=1012.686,-122.315,394.726,164.629,68.781,162.278
C00661=1012.687,-122.703,394.754,164.617,68.677,162.249
C00662=1012.690,-123.091,394.782,164.605,68.573,162.220
C00663=1012.691,-123.479,394.810,164.593,68.468,162.192
C00664=1012.693,-123.868,394.839,164.581,68.363,162.163
C00665=1012.695,-124.256,394.867,164.570,68.256,162.134
C00666=1012.697,-124.645,394.896,164.559,68.148,162.106
C00667=1012.700,-125.033,394.924,164.548,68.039,162.077
C00668=1012.701,-125.421,394.952,164.537,67.929,162.047
C00669=1012.704,-125.809,394.980,164.527,67.818,162.019
C00670=1012.706,-126.198,395.009,164.517,67.706,161.990
C00671=1012.708,-126.586,395.037,164.507,67.595,161.961
C00672=1012.709,-126.974,395.066,164.497,67.481,161.932
C00673=1012.712,-127.362,395.094,164.487,67.366,161.904
C00674=1012.714,-127.750,395.123,164.479,67.250,161.875
C00675=1012.716,-128.138,395.151,164.470,67.133,161.846
C00676=1012.718,-128.527,395.180,164.460,67.015,161.817
C00677=1012.721,-128.915,395.208,164.453,66.896,161.789
C00678=1012.723,-129.302,395.237,164.444,66.775,161.759
C00679=1012.725,-129.691,395.266,164.436,66.655,161.730
C00680=1012.727,-130.079,395.294,164.428,66.532,161.701
C00681=1012.730,-130.467,395.323,164.421,66.409,161.672
C00682=1012.733,-130.855,395.351,164.414,66.285,161.644
C00683=1012.735,-131.244,395.380,164.407,66.159,161.615
C00684=1012.737,-131.634,395.409,164.401,66.031,161.586
C00685=1012.740,-132.020,395.438,164.395,65.904,161.557
C00686=1012.743,-132.407,395.466,164.388,65.775,161.527
C00687=1012.746,-132.796,395.495,164.383,65.644,161.498
C00688=1012.748,-133.183,395.524,164.378,65.513,161.469
C00689=1012.751,-133.572,395.553,164.372,65.380,161.440
C00690=1012.753,-133.960,395.581,164.367,65.246,161.411
C00691=1012.820,13.706,384.977,165.533,60.683,160.899
C00692=1012.819,13.328,385.007,165.526,60.761,160.913
C00693=1012.817,12.944,385.036,165.519,60.839,160.927
C00694=1012.816,12.559,385.066,165.511,60.918,160.940
C00695=1012.814,12.177,385.096,165.504,60.995,160.954
C00696=1012.813,11.805,385.125,165.497,61.071,160.967
C00697=1012.812,11.441,385.153,165.491,61.144,160.980
C00698=1012.810,11.076,385.182,165.485,61.216,160.993
C00699=1012.809,10.702,385.210,165.478,61.290,161.006
C00700=1012.808,10.324,385.239,165.472,61.365,161.019
C00701=1012.806,9.948,385.269,165.465,61.438,161.032
C00702=1012.805,9.573,385.299,165.460,61.511,161.045
C00703=1012.804,9.199,385.327,165.454,61.583,161.058
C00704=1012.802,8.825,385.356,165.447,61.655,161.070
C00705=1012.802,8.451,385.385,165.441,61.727,161.083
C00706=1012.800,8.075,385.414,165.435,61.798,161.096
C00707=1012.799,7.697,385.443,165.430,61.868,161.109
C00708=1012.797,7.315,385.474,165.423,61.940,161.121
C00709=1012.796,6.929,385.503,165.418,62.012,161.135
C00710=1012.795,6.538,385.533,165.413,62.083,161.148
C00711=1012.794,6.145,385.564,165.407,62.156,161.161
C00712=1012.793,5.752,385.594,165.402,62.227,161.174
C00713=1012.791,5.362,385.624,165.396,62.298,161.186
C00714=1012.790,4.973,385.655,165.391,62.367,161.199
C00715=1012.788,4.583,385.685,165.386,62.437,161.212
C00716=1012.788,4.192,385.715,165.381,62.505,161.224
C00717=1012.787,3.820,385.744,165.376,62.571,161.236
C00718=1012.785,3.475,385.771,165.372,62.631,161.248
C00719=1012.784,3.152,385.796,165.367,62.687,161.257
C00720=1012.783,2.828,385.821,165.364,62.742,161.268
C00721=1012.783,2.486,385.848,165.359,62.800,161.278
C00722=1012.781,2.115,385.876,165.356,62.863,161.290
C00723=1012.780,1.723,385.907,165.351,62.929,161.302
C00724=1012.779,1.325,385.937,165.347,62.996,161.315
C00725=1012.778,0.928,385.968,165.342,63.061,161.327
C00726=1012.777,0.534,385.999,165.338,63.125,161.339
C00727=1012.776,0.139,386.029,165.333,63.190,161.351
C00728=1012.775,-0.259,386.060,165.329,63.254,161.363
C00729=1012.774,-0.659,386.091,165.326,63.318,161.375
C00730=1012.773,-1.062,386.122,165.321,63.382,161.387
C00731=1012.772,-1.467,386.153,165.317,63.445,161.399
C00732=1012.771,-1.873,386.184,165.313,63.508,161.411
C00733=1012.770,-2.282,386.216,165.309,63.572,161.423
C00734=1012.769,-2.693,386.248,165.305,63.634,161.435
C00735=1012.768,-3.104,386.280,165.302,63.696,161.447
C00736=1012.766,-3.506,386.310,165.299,63.757,161.459
C00737=1012.765,-3.892,386.341,165.295,63.813,161.469
C00738=1012.765,-4.271,386.370,165.292,63.869,161.480
C00739=1012.764,-4.662,386.401,165.288,63.926,161.491
C00740=1012.763,-5.077,386.433,165.284,63.986,161.502
C00741=1012.762,-5.291,386.449,165.283,64.016,161.508
C00742=1012.762,-5.507,386.466,165.281,64.047,161.514
C00743=1012.761,-5.724,386.483,165.280,64.077,161.520
C00744=1012.761,-5.941,386.499,165.278,64.108,161.526
C00745=1012.760,-6.158,386.516,165.277,64.139,161.532
C00746=1012.760,-6.375,386.533,165.275,64.169,161.538
C00747=1012.760,-6.590,386.550,165.273,64.198,161.543
C00748=1012.759,-6.807,386.566,165.271,64.228,161.549
C00749=1012.758,-7.022,386.582,165.271,64.257,161.555
C00750=1012.758,-7.236,386.599,165.268,64.286,161.560
C00751=1012.757,-7.449,386.616,165.267,64.315,161.566
C00752=1012.757,-7.663,386.632,165.265,64.343,161.571
C00753=1012.757,-7.875,386.649,165.264,64.372,161.577
C00754=1012.756,-8.088,386.665,165.262,64.400,161.583
C00755=1012.756,-8.298,386.682,165.260,64.428,161.588
C00756=1012.755,-8.510,386.698,165.259,64.455,161.593
C00757=1012.755,-8.721,386.714,165.258,64.483,161.599
C00758=1012.755,-8.932,386.730,165.256,64.511,161.604
C00759=1012.754,-9.143,386.747,165.255,64.538,161.609
C00760=1012.753,-9.565,386.779,165.252,64.592,161.620
C00761=1012.752,-9.987,386.812,165.250,64.644,161.630
C00762=1012.752,-10.407,386.844,165.248,64.697,161.641
C00763=1012.751,-10.826,386.877,165.243,64.748,161.650
C00764=1012.750,-11.244,386.909,165.242,64.798,161.661
C00765=1012.749,-11.660,386.941,165.239,64.849,161.670
C00766=1012.749,-12.075,386.974,165.237,64.897,161.680
C00767=1012.748,-12.489,387.005,165.235,64.945,161.690
C00768=1012.747,-12.897,387.037,165.232,64.993,161.699
C00769=1012.746,-13.296,387.068,165.230,65.038,161.708
C00770=1012.745,-13.683,387.098,165.228,65.081,161.717
C00771=1012.745,-14.062,387.127,165.227,65.123,161.725
C00772=1012.745,-14.436,387.156,165.224,65.163,161.733
C00773=1012.744,-14.812,387.184,165.222,65.204,161.741
C00774=1012.743,-15.196,387.215,165.220,65.245,161.749
C00775=1012.743,-15.588,387.245,165.218,65.285,161.757
C00776=1012.742,-15.984,387.276,165.217,65.326,161.765
C00777=1012.741,-16.380,387.306,165.213,65.366,161.773
C00778=1012.741,-16.778,387.337,165.212,65.406,161.781
C00779=1012.741,-17.174,387.367,165.210,65.445,161.789
C00780=1012.740,-17.560,387.397,165.208,65.482,161.796
C00781=1012.739,-17.763,387.413,165.207,65.502,161.800
C00782=1012.739,-17.990,387.430,165.207,65.523,161.805
C00783=1012.739,-18.242,387.450,165.205,65.547,161.809
C00784=1012.739,-18.515,387.471,165.204,65.572,161.814
C00785=1012.738,-18.795,387.492,165.202,65.598,161.819
C00786=1012.738,-19.069,387.513,165.200,65.623,161.824
C00787=1012.738,-19.325,387.534,165.200,65.645,161.829
C00788=1012.737,-19.556,387.551,165.199,65.666,161.833
C00789=1012.737,-19.761,387.567,165.198,65.684,161.836
C00790=1012.737,-20.112,387.595,165.196,65.715,161.842
C00791=1012.736,-20.509,387.625,165.195,65.748,161.849
C00792=1012.736,-20.902,387.655,165.193,65.781,161.856
C00793=1012.735,-21.296,387.686,165.192,65.813,161.862
C00794=1012.735,-21.689,387.716,165.189,65.845,161.868
C00795=1012.734,-22.083,387.747,165.188,65.876,161.875
C00796=1012.734,-22.476,387.777,165.186,65.907,161.881
C00797=1012.734,-22.869,387.807,165.185,65.936,161.887
C00798=1012.733,-23.263,387.838,165.183,65.965,161.892
C00799=1012.733,-23.656,387.868,165.181,65.994,161.898
C00800=1012.732,-24.050,387.899,165.180,66.022,161.903
C00801=1012.732,-24.443,387.929,165.178,66.049,161.909
C00802=1012.732,-24.836,387.959,165.176,66.076,161.914
C00803=1012.731,-25.230,387.990,165.174,66.102,161.919
C00804=1012.731,-25.623,388.020,165.172,66.127,161.924
C00805=1012.730,-26.017,388.051,165.171,66.152,161.929
C00806=1012.730,-26.410,388.081,165.169,66.177,161.933
C00807=1012.730,-26.803,388.111,165.167,66.199,161.938
C00808=1012.729,-27.197,388.142,165.165,66.222,161.942
C00809=1012.729,-27.590,388.172,165.165,66.245,161.947
C00810=1012.729,-27.984,388.203,165.163,66.266,161.951
C00811=1012.729,-28.378,388.233,165.160,66.287,161.954
C00812=1012.728,-28.772,388.263,165.159,66.307,161.958
C00813=1012.728,-29.165,388.294,165.157,66.328,161.962
C00814=1012.728,-29.558,388.324,165.156,66.347,161.966
C00815=1012.728,-29.952,388.355,165.154,66.365,161.969
C00816=1012.728,-30.346,388.385,165.152,66.383,161.972
C00817=1012.727,-30.739,388.416,165.151,66.400,161.975
C00818=1012.727,-31.133,388.445,165.149,66.416,161.978
C00819=1012.727,-31.527,388.477,165.147,66.432,161.981
C00820=1012.727,-31.920,388.507,165.144,66.447,161.983
C00821=1012.727,-32.314,388.537,165.143,66.462,161.986
C00822=1012.726,-32.707,388.568,165.140,66.476,161.988
C00823=1012.727,-33.101,388.599,165.139,66.489,161.990
C00824=1012.726,-33.495,388.628,165.137,66.502,161.992
C00825=1012.726,-33.889,388.659,165.136,66.514,161.994
C00826=1012.727,-34.282,388.690,165.133,66.525,161.996
C00827=1012.726,-34.676,388.720,165.131,66.536,161.997
C00828=1012.726,-35.069,388.750,165.129,66.545,161.998
C00829=1012.726,-35.463,388.780,165.126,66.555,162.000
C00830=1012.726,-35.857,388.811,165.124,66.563,162.001
C00831=1012.726,-36.250,388.841,165.122,66.572,162.002
C00832=1012.726,-36.643,388.872,165.120,66.579,162.002
C00833=1012.726,-37.037,388.903,165.118,66.586,162.003
C00834=1012.725,-37.430,388.933,165.117,66.592,162.004
C00835=1012.726,-37.825,388.963,165.114,66.597,162.004
C00836=1012.725,-38.218,388.994,165.111,66.602,162.004
C00837=1012.725,-38.611,389.024,165.110,66.606,162.004
C00838=1012.726,-39.005,389.055,165.108,66.609,162.004
C00839=1012.726,-39.398,389.085,165.106,66.612,162.004
C00840=1012.726,-39.791,389.115,165.103,66.614,162.003
C00841=1012.726,-40.185,389.146,165.101,66.615,162.002
C00842=1012.725,-40.579,389.177,165.099,66.616,162.002
C00843=1012.725,-40.972,389.207,165.096,66.616,162.001
C00844=1012.726,-41.366,389.237,165.093,66.615,161.999
C00845=1012.726,-41.759,389.267,165.091,66.614,161.998
C00846=1012.727,-42.152,389.298,165.089,66.612,161.997
C00847=1012.726,-42.545,389.328,165.086,66.610,161.995
C00848=1012.726,-42.939,389.359,165.083,66.606,161.993
C00849=1012.727,-43.332,389.390,165.082,66.602,161.991
C00850=1012.727,-43.725,389.420,165.078,66.598,161.989
C00851=1012.726,-44.118,389.450,165.076,66.592,161.987
C00852=1012.728,-44.511,389.481,165.074,66.586,161.984
C00853=1012.727,-44.904,389.511,165.071,66.580,161.982
C00854=1012.727,-45.297,389.541,165.069,66.572,161.979
C00855=1012.728,-45.690,389.573,165.065,66.564,161.976
C00856=1012.728,-46.083,389.602,165.063,66.555,161.973
C00857=1012.728,-46.476,389.633,165.060,66.546,161.970
C00858=1012.728,-46.869,389.664,165.056,66.536,161.966
C00859=1012.728,-47.262,389.694,165.053,66.525,161.962
C00860=1012.729,-47.655,389.724,165.051,66.514,161.959
C00861=1012.729,-48.048,389.754,165.049,66.502,161.955
C00862=1012.730,-48.441,389.784,165.045,66.489,161.951
C00863=1012.730,-48.833,389.816,165.042,66.475,161.947
C00864=1012.730,-49.226,389.846,165.040,66.461,161.943
C00865=1012.730,-49.619,389.876,165.036,66.446,161.937
C00866=1012.731,-50.012,389.906,165.034,66.431,161.934
C00867=1012.731,-50.405,389.937,165.030,66.415,161.928
C00868=1012.731,-50.797,389.967,165.028,66.397,161.923
C00869=1012.732,-51.190,389.998,165.024,66.380,161.918
C00870=1012.732,-51.583,390.028,165.021,66.362,161.913
C00871=1012.733,-51.976,390.059,165.018,66.343,161.907
C00872=1012.733,-52.368,390.089,165.015,66.323,161.902
C00873=1012.733,-52.761,390.120,165.013,66.303,161.896
C00874=1012.734,-53.154,390.150,165.009,66.281,161.890
C00875=1012.735,-53.546,390.180,165.005,66.260,161.884
C00876=1012.735,-53.940,390.211,165.003,66.238,161.878
C00877=1012.735,-54.331,390.241,165.000,66.214,161.872
C00878=1012.737,-54.724,390.272,164.996,66.191,161.865
C00879=1012.736,-55.117,390.302,164.994,66.166,161.859
C00880=1012.737,-55.510,390.332,164.991,66.141,161.852
C00881=1012.737,-55.903,390.363,164.987,66.115,161.844
C00882=1012.739,-56.296,390.393,164.984,66.088,161.837
C00883=1012.738,-56.689,390.424,164.980,66.061,161.830
C00884=1012.739,-57.082,390.454,164.978,66.033,161.823
C00885=1012.740,-57.476,390.485,164.974,66.004,161.815
C00886=1012.740,-57.871,390.516,164.971,65.974,161.807
C00887=1012.741,-58.266,390.546,164.968,65.944,161.799
C00888=1012.741,-58.661,390.577,164.964,65.913,161.791
C00889=1012.742,-59.058,390.607,164.961,65.880,161.783
C00890=1012.743,-59.454,390.638,164.957,65.848,161.774
C00891=1012.744,-59.850,390.669,164.954,65.815,161.766
C00892=1012.744,-60.248,390.700,164.951,65.781,161.757
C00893=1012.745,-60.646,390.731,164.947,65.746,161.748
C00894=1012.746,-61.045,390.762,164.945,65.711,161.740
C00895=1012.747,-61.443,390.793,164.941,65.674,161.730
C00896=1012.747,-61.843,390.824,164.938,65.637,161.721
C00897=1012.748,-62.243,390.854,164.935,65.599,161.712
C00898=1012.749,-62.643,390.886,164.931,65.560,161.702
C00899=1012.749,-63.045,390.916,164.928,65.521,161.692
C00900=1012.751,-63.446,390.947,164.925,65.480,161.682
C00901=1012.751,-63.848,390.979,164.921,65.439,161.672
C00902=1012.752,-64.250,391.010,164.918,65.397,161.662
C00903=1012.753,-64.652,391.042,164.915,65.355,161.651
C00904=1012.753,-65.056,391.073,164.912,65.311,161.641
C00905=1012.755,-65.458,391.104,164.910,65.267,161.631
C00906=1012.756,-65.861,391.135,164.906,65.222,161.620
C00907=1012.756,-66.266,391.167,164.903,65.176,161.609
C00908=1012.758,-66.670,391.198,164.900,65.129,161.597
C00909=1012.758,-67.074,391.229,164.897,65.082,161.586
C00910=1012.760,-67.477,391.261,164.894,65.034,161.575
C00911=1012.760,-67.882,391.292,164.891,64.986,161.564
C00912=1012.761,-68.287,391.323,164.888,64.936,161.552
C00913=1012.763,-68.690,391.355,164.885,64.886,161.540
C00914=1012.763,-69.095,391.386,164.882,64.834,161.528
C00915=1012.765,-69.500,391.418,164.879,64.783,161.516
C00916=1012.766,-69.904,391.449,164.877,64.730,161.504
C00917=1012.767,-70.309,391.480,164.874,64.677,161.492
C00918=1012.768,-70.713,391.511,164.871,64.623,161.479
C00919=1012.769,-71.118,391.543,164.869,64.568,161.467
C00920=1012.770,-71.522,391.574,164.865,64.513,161.454
C00921=1012.771,-71.926,391.606,164.862,64.456,161.441
C00922=1012.773,-72.330,391.637,164.860,64.399,161.429
C00923=1012.774,-72.734,391.669,164.858,64.341,161.416
C00924=1012.776,-73.138,391.699,164.855,64.283,161.403
C00925=1012.777,-73.541,391.731,164.853,64.224,161.390
C00926=1012.778,-73.945,391.762,164.851,64.164,161.376
C00927=1012.778,-74.348,391.793,164.849,64.103,161.363
C00928=1012.780,-74.751,391.825,164.847,64.042,161.349
C00929=1012.781,-75.155,391.856,164.845,63.979,161.336
C00930=1012.783,-75.557,391.887,164.842,63.916,161.322
C00931=1012.784,-75.961,391.919,164.841,63.853,161.308
C00932=1012.786,-76.364,391.950,164.839,63.789,161.294
C00933=1012.787,-76.766,391.981,164.836,63.724,161.280
C00934=1012.788,-77.168,392.012,164.835,63.658,161.266
C00935=1012.789,-77.569,392.043,164.834,63.592,161.252
C00936=1012.791,-77.972,392.074,164.832,63.525,161.238
C00937=1012.793,-78.373,392.105,164.830,63.456,161.223
C00938=1012.794,-78.774,392.137,164.828,63.388,161.209
C00939=1012.796,-79.174,392.167,164.827,63.319,161.194
C00940=1012.797,-79.574,392.199,164.827,63.249,161.180
C00941=1012.798,-79.974,392.230,164.826,63.179,161.165
C00942=1012.800,-80.373,392.261,164.824,63.108,161.151
C00943=1012.801,-80.771,392.292,164.823,63.037,161.136
C00944=1012.803,-81.168,392.322,164.822,62.965,161.121
C00945=1012.804,-81.566,392.353,164.821,62.892,161.106
C00946=1012.806,-81.964,392.384,164.821,62.818,161.091
C00947=1012.808,-82.363,392.415,164.820,62.743,161.076
C00948=1012.810,-82.759,392.446,164.820,62.669,161.061
C00949=1012.811,-83.156,392.477,164.819,62.593,161.045
C00950=1012.813,-83.552,392.507,164.819,62.517,161.030
C00951=1012.815,-83.944,392.537,164.818,62.441,161.015
C00952=1012.816,-84.336,392.567,164.818,62.364,160.999
C00953=1012.818,-84.754,392.600,164.818,62.282,160.983
C00954=1012.819,-84.985,392.618,164.818,62.236,160.974
C00955=1012.820,-85.222,392.637,164.819,62.188,160.965
C00956=1012.821,-85.462,392.655,164.819,62.140,160.955
C00957=1012.822,-85.697,392.673,164.820,62.093,160.946
C00958=1012.823,-85.919,392.690,164.819,62.047,160.937
C00959=1012.825,-86.327,392.721,164.820,61.964,160.921
C00960=1012.827,-86.715,392.752,164.821,61.883,160.905
C00961=1012.829,-87.093,392.781,164.821,61.805,160.890
C00962=1012.831,-87.460,392.809,164.821,61.728,160.875
C00963=1012.833,-87.823,392.838,164.824,61.652,160.860
C00964=1012.834,-88.200,392.867,164.824,61.572,160.845
C00965=1012.836,-88.585,392.896,164.825,61.489,160.829
C00966=1012.837,-88.804,392.913,164.826,61.441,160.820
C00967=1012.838,-89.046,392.932,164.827,61.389,160.810
C00968=1012.840,-89.302,392.952,164.828,61.333,160.800
C00969=1012.841,-89.561,392.972,164.828,61.277,160.789
C00970=1012.842,-89.812,392.991,164.829,61.221,160.778
C00971=1012.843,-90.071,393.011,164.831,61.164,160.768
C00972=1012.610,-133.983,395.183,165.422,73.776,163.914
C00973=1012.608,-133.594,395.153,165.467,73.917,163.978
C00974=1012.606,-133.207,395.124,165.512,74.058,164.042
C00975=1012.604,-132.819,395.095,165.558,74.198,164.107
C00976=1012.602,-132.431,395.065,165.605,74.336,164.172
C00977=1012.601,-132.043,395.036,165.654,74.474,164.239
C00978=1012.599,-131.655,395.007,165.703,74.612,164.306
C00979=1012.597,-131.267,394.977,165.754,74.749,164.375
C00980=1012.595,-130.879,394.948,165.807,74.885,164.445
C00981=1012.593,-130.491,394.919,165.860,75.021,164.515
C00982=1012.592,-130.103,394.889,165.913,75.156,164.585
C00983=1012.590,-129.715,394.860,165.968,75.291,164.657
C00984=1012.588,-129.327,394.830,166.024,75.424,164.730
C00985=1012.587,-128.939,394.801,166.082,75.558,164.804
C00986=1012.585,-128.551,394.772,166.141,75.690,164.880
C00987=1012.583,-128.163,394.742,166.201,75.822,164.955
C00988=1012.582,-127.775,394.713,166.262,75.954,165.033
C00989=1012.580,-127.387,394.684,166.324,76.085,165.110
C00990=1012.579,-126.999,394.654,166.386,76.214,165.189
C00991=1012.578,-126.610,394.624,166.452,76.344,165.270
C00992=1012.577,-126.222,394.595,166.517,76.473,165.351
C00993=1012.574,-125.834,394.565,166.585,76.601,165.434
C00994=1012.573,-125.446,394.536,166.653,76.729,165.518
C00995=1012.571,-125.058,394.506,166.725,76.856,165.604
C00996=1012.570,-124.669,394.477,166.797,76.983,165.690
C00997=1012.569,-124.281,394.448,166.869,77.109,165.777
C00998=1012.568,-123.893,394.418,166.944,77.234,165.867
C00999=1012.566,-123.505,394.389,167.020,77.359,165.957
C01000=1012.564,-123.116,394.359,167.098,77.484,166.049
C01001=1012.563,-122.728,394.330,167.177,77.607,166.142
C01002=1012.561,-122.340,394.300,167.259,77.730,166.238
C01003=1012.561,-121.952,394.270,167.341,77.853,166.334
C01004=1012.559,-121.564,394.241,167.426,77.975,166.432
C01005=1012.559,-121.176,394.211,167.512,78.097,166.532
C01006=1012.557,-120.787,394.182,167.598,78.217,166.632
C01007=1012.556,-120.399,394.152,167.688,78.337,166.734
C01008=1012.555,-120.011,394.123,167.778,78.457,166.838
C01009=1012.554,-119.622,394.093,167.871,78.576,166.944
C01010=1012.552,-119.234,394.064,167.968,78.695,167.053
C01011=1012.551,-118.845,394.035,168.065,78.813,167.162
C01012=1012.550,-118.457,394.004,168.162,78.931,167.273
C01013=1012.549,-118.069,393.974,168.264,79.047,167.386
C01014=1012.548,-117.680,393.945,168.366,79.163,167.501
C01015=1012.547,-117.291,393.915,168.471,79.279,167.618
C01016=1012.545,-116.903,393.886,168.580,79.395,167.739
C01017=1012.545,-116.515,393.856,168.690,79.509,167.860
C01018=1012.544,-116.126,393.827,168.800,79.623,167.982
C01019=1012.543,-115.737,393.797,168.914,79.737,168.108
C01020=1012.542,-115.349,393.768,169.029,79.849,168.235
C01021=1012.541,-114.961,393.738,169.148,79.962,168.365
C01022=1012.540,-114.573,393.708,169.271,80.074,168.499
C01023=1012.539,-114.184,393.678,169.393,80.186,168.633
C01024=1012.538,-113.795,393.649,169.519,80.295,168.770
C01025=1012.537,-113.406,393.619,169.647,80.406,168.909
C01026=1012.536,-113.018,393.590,169.780,80.516,169.052
C01027=1012.535,-112.629,393.560,169.915,80.624,169.197
C01028=1012.535,-112.240,393.530,170.052,80.733,169.346
C01029=1012.534,-111.851,393.501,170.192,80.841,169.496
C01030=1012.533,-111.463,393.471,170.337,80.948,169.651
C01031=1012.532,-111.073,393.441,170.481,81.054,169.806
C01032=1012.531,-110.685,393.410,170.631,81.161,169.966
C01033=1012.530,-110.296,393.381,170.782,81.266,170.127
C01034=1012.529,-109.908,393.351,170.938,81.371,170.293
C01035=1012.529,-109.519,393.321,171.100,81.476,170.464
C01036=1012.528,-109.124,393.291,171.264,81.581,170.639
C01037=1012.527,-108.707,393.260,171.445,81.691,170.829
C01038=1012.527,-108.488,393.242,171.540,81.750,170.930
C01039=1012.527,-108.263,393.225,171.636,81.808,171.032
C01040=1012.526,-108.032,393.207,171.741,81.868,171.142
C01041=1012.525,-107.801,393.190,171.847,81.929,171.253
C01042=1012.525,-107.568,393.172,171.950,81.989,171.362
C01043=1012.524,-107.338,393.154,172.056,82.049,171.474
C01044=1012.524,-107.112,393.137,172.165,82.108,171.588
C01045=1012.524,-106.891,393.120,172.269,82.165,171.697
C01046=1012.524,-106.677,393.104,172.373,82.220,171.806
C01047=1012.523,-106.270,393.072,172.573,82.324,172.016
C01048=1012.522,-105.879,393.042,172.771,82.423,172.223
C01049=1012.521,-105.490,393.013,172.972,82.521,172.432
C01050=1012.520,-105.102,392.983,173.175,82.618,172.644
C01051=1012.520,-104.714,392.953,173.384,82.716,172.861
C01052=1012.520,-104.325,392.924,173.600,82.812,173.086
C01053=1012.519,-103.937,392.893,173.819,82.907,173.312
C01054=1012.519,-103.551,392.863,174.039,83.002,173.541
C01055=1012.518,-103.164,392.834,174.268,83.095,173.778
C01056=1012.518,-102.778,392.804,174.503,83.189,174.022
C01057=1012.516,-102.393,392.775,174.742,83.282,174.268
C01058=1012.517,-102.008,392.745,174.983,83.373,174.517
C01059=1012.516,-101.625,392.716,175.232,83.464,174.774
C01060=1012.515,-101.242,392.686,175.485,83.554,175.034
C01061=1012.515,-100.860,392.657,175.745,83.643,175.302
C01062=1012.515,-100.479,392.628,176.008,83.731,175.573
C01063=1012.514,-100.100,392.598,176.281,83.819,175.853
C01064=1012.513,-99.722,392.569,176.557,83.905,176.136
C01065=1012.513,-99.344,392.540,176.835,83.990,176.422
C01066=1012.512,-98.967,392.510,177.124,84.074,176.717
C01067=1012.512,-98.591,392.482,177.421,84.159,177.021
C01068=1012.512,-98.215,392.453,177.722,84.242,177.328
C01069=1012.512,-97.839,392.424,178.026,84.324,177.640
C01070=1012.512,-97.463,392.395,178.346,84.407,177.966
C01071=1012.510,-97.088,392.366,178.664,84.487,178.291
C01072=1012.510,-96.711,392.337,179.000,84.568,178.633
C01073=1012.510,-96.335,392.309,179.338,84.648,178.978
C01074=1012.509,-95.957,392.279,179.688,84.728,179.334
C01075=1012.509,-95.579,392.250,-179.957,84.806,179.695
C01076=1012.508,-95.200,392.220,-179.584,84.885,-179.925
C01077=1012.509,-94.819,392.191,-179.205,84.962,-179.541
C01078=1012.508,-94.437,392.162,-178.814,85.040,-179.143
C01079=1012.508,-94.055,392.132,-178.418,85.117,-178.741
C01080=1012.507,-93.671,392.102,-178.009,85.193,-178.325
C01081=1012.507,-93.286,392.073,-177.576,85.269,-177.887
C01082=1012.506,-92.900,392.043,-177.147,85.344,-177.451
C01083=1012.507,-92.512,392.013,-176.693,85.419,-176.992
C01084=1012.506,-92.125,391.984,-176.233,85.492,-176.526
C01085=1012.506,-91.737,391.953,-175.757,85.565,-176.045
C01086=1012.506,-91.348,391.923,-175.274,85.638,-175.555
C01087=1012.505,-90.960,391.893,-174.764,85.710,-175.040
C01088=1012.505,-90.605,391.866,-174.298,85.775,-174.569
C01089=1012.505,-90.336,391.846,-173.937,85.822,-174.204
C01090=1012.504,-90.126,391.828,-173.643,85.861,-173.907
C01091=1012.505,-89.892,391.811,-173.321,85.902,-173.582
C01092=1012.505,-89.641,391.791,-172.959,85.946,-173.216
C01093=1012.504,-89.382,391.771,-172.587,85.992,-172.841
C01094=1012.504,-88.980,391.740,-171.990,86.061,-172.239
C01095=1012.504,-88.664,391.716,-171.520,86.114,-171.764
C01096=1012.503,-88.280,391.686,-170.921,86.179,-171.161
C01097=1012.503,-87.903,391.656,-170.314,86.242,-170.549
C01098=1012.503,-87.541,391.629,-169.727,86.301,-169.956
C01099=1012.503,-87.172,391.601,-169.105,86.361,-169.330
C01100=1012.503,-86.795,391.571,-168.462,86.421,-168.682
C01101=1012.503,-86.408,391.541,-167.780,86.482,-167.995
C01102=1012.502,-86.000,391.509,-167.042,86.544,-167.251
C01103=1012.502,-85.777,391.492,-166.623,86.578,-166.831
C01104=1012.502,-85.543,391.474,-166.178,86.613,-166.383
C01105=1012.502,-85.303,391.455,-165.723,86.649,-165.925
C01106=1012.502,-85.065,391.436,-165.258,86.684,-165.457
C01107=1012.502,-84.835,391.419,-164.800,86.717,-164.997
C01108=1012.502,-84.417,391.387,-163.966,86.777,-164.157
C01109=1012.502,-84.024,391.357,-163.139,86.832,-163.326
C01110=1012.501,-83.633,391.327,-162.302,86.886,-162.485
C01111=1012.501,-83.238,391.296,-161.451,86.938,-161.629
C01112=1012.501,-82.841,391.265,-160.553,86.991,-160.727
C01113=1012.501,-82.445,391.234,-159.639,87.042,-159.808
C01114=1012.501,-82.046,391.203,-158.698,87.091,-158.863
C01115=1012.501,-81.647,391.172,-157.740,87.140,-157.901
C01116=1012.501,-81.250,391.141,-156.755,87.187,-156.911
C01117=1012.501,-80.853,391.110,-155.735,87.233,-155.888
C01118=1012.500,-80.455,391.080,-154.706,87.277,-154.854
C01119=1012.500,-80.057,391.049,-153.642,87.321,-153.786
C01120=1012.500,-79.656,391.018,-152.542,87.363,-152.683
C01121=1012.500,-79.256,390.987,-151.427,87.404,-151.563
C01122=1012.499,-78.856,390.956,-150.282,87.444,-150.415
C01123=1012.500,-78.455,390.925,-149.131,87.481,-149.260
C01124=1012.500,-78.054,390.894,-147.944,87.518,-148.070
C01125=1012.500,-77.653,390.863,-146.722,87.553,-146.844
C01126=1012.499,-77.251,390.831,-145.496,87.587,-145.614
C01127=1012.499,-76.849,390.800,-144.234,87.619,-144.349
C01128=1012.500,-76.446,390.769,-142.972,87.649,-143.082
C01129=1012.499,-76.043,390.738,-141.676,87.679,-141.783
C01130=1012.499,-75.641,390.706,-140.346,87.707,-140.450
C01131=1012.499,-75.238,390.675,-139.020,87.733,-139.120
C01132=1012.498,-74.835,390.644,-137.663,87.758,-137.760
C01133=1012.499,-74.431,390.612,-136.312,87.781,-136.406
C01134=1012.498,-74.028,390.582,-134.934,87.802,-135.024
C01135=1012.499,-73.625,390.550,-133.542,87.822,-133.629
C01136=1012.498,-73.222,390.519,-132.149,87.841,-132.232
C01137=1012.498,-72.818,390.487,-130.747,87.858,-130.828
C01138=1012.499,-72.414,390.456,-129.348,87.874,-129.425
C01139=1012.499,-72.010,390.425,-127.944,87.888,-128.018
C01140=1012.498,-71.606,390.393,-126.522,87.900,-126.594
C01141=1012.498,-71.202,390.362,-125.108,87.912,-125.176
C01142=1012.498,-70.798,390.331,-123.695,87.922,-123.761
C01143=1012.498,-70.393,390.299,-122.312,87.930,-122.375
C01144=1012.498,-69.989,390.268,-120.918,87.937,-120.979
C01145=1012.498,-69.585,390.236,-119.540,87.943,-119.597
C01146=1012.498,-69.180,390.205,-118.172,87.948,-118.226
C01147=1012.498,-68.776,390.174,-116.799,87.951,-116.850
C01148=1012.498,-68.372,390.142,-115.464,87.953,-115.513
C01149=1012.497,-67.967,390.111,-114.146,87.954,-114.193
C01150=1012.498,-67.562,390.080,-112.831,87.955,-112.875
C01151=1012.498,-67.159,390.048,-111.556,87.953,-111.597
C01152=1012.498,-66.754,390.017,-110.282,87.951,-110.322
C01153=1012.498,-66.351,389.985,-109.035,87.948,-109.072
C01154=1012.497,-65.947,389.954,-107.811,87.944,-107.846
C01155=1012.498,-65.544,389.922,-106.615,87.939,-106.647
C01156=1012.498,-65.141,389.891,-105.444,87.934,-105.474
C01157=1012.497,-64.739,389.860,-104.302,87.928,-104.329
C01158=1012.498,-64.336,389.829,-103.186,87.921,-103.211
C01159=1012.498,-63.934,389.797,-102.099,87.913,-102.122
C01160=1012.498,-63.532,389.767,-101.040,87.904,-101.062
C01161=1012.498,-63.131,389.736,-100.010,87.896,-100.029
C01162=1012.497,-62.730,389.704,-98.989,87.886,-99.006
C01163=1012.498,-62.330,389.674,-98.016,87.877,-98.030
C01164=1012.498,-61.930,389.643,-97.053,87.867,-97.065
C01165=1012.498,-61.530,389.611,-96.138,87.856,-96.149
C01166=1012.498,-61.132,389.580,-95.250,87.845,-95.259
C01167=1012.498,-60.733,389.549,-94.371,87.834,-94.377
C01168=1012.498,-60.335,389.519,-93.521,87.823,-93.526
C01169=1012.498,-59.938,389.487,-92.717,87.811,-92.720
C01170=1012.498,-59.540,389.456,-91.922,87.799,-91.923
C01171=1012.498,-59.144,389.426,-91.135,87.787,-91.134
C01172=1012.497,-58.748,389.395,-90.408,87.776,-90.405
C01173=1012.498,-58.353,389.364,-89.693,87.763,-89.689
C01174=1012.497,-57.958,389.333,-89.001,87.751,-88.995
C01175=1012.498,-57.564,389.304,-88.336,87.739,-88.329
C01176=1012.497,-57.170,389.273,-87.693,87.727,-87.684
C01177=1012.497,-56.777,389.242,-87.057,87.715,-87.046
C01178=1012.497,-56.384,389.212,-86.447,87.702,-86.435
C01179=1012.497,-55.990,389.181,-85.876,87.690,-85.862
C01180=1012.497,-55.598,389.150,-85.311,87.678,-85.296
C01181=1012.498,-55.205,389.120,-84.784,87.666,-84.768
C01182=1012.497,-54.813,389.090,-84.262,87.654,-84.245
C01183=1012.497,-54.420,389.059,-83.759,87.643,-83.740
C01184=1012.497,-54.028,389.028,-83.266,87.631,-83.246
C01185=1012.497,-53.635,388.998,-82.803,87.620,-82.781
C01186=1012.497,-53.243,388.967,-82.350,87.609,-82.327
C01187=1012.497,-52.850,388.937,-81.932,87.598,-81.908
C01188=1012.497,-52.457,388.906,-81.500,87.587,-81.474
C01189=1012.497,-52.065,388.876,-81.118,87.576,-81.092
C01190=1012.497,-51.672,388.846,-80.723,87.566,-80.695
C01191=1012.497,-51.280,388.815,-80.378,87.556,-80.349
C01192=1012.496,-50.886,388.785,-80.018,87.547,-79.987
C01193=1012.497,-50.494,388.754,-79.695,87.537,-79.664
C01194=1012.496,-50.101,388.724,-79.358,87.527,-79.326
C01195=1012.497,-49.708,388.694,-79.063,87.519,-79.029
C01196=1012.497,-49.316,388.663,-78.775,87.510,-78.741
C01197=1012.497,-48.923,388.633,-78.501,87.502,-78.465
C01198=1012.497,-48.530,388.602,-78.245,87.494,-78.209
C01199=1012.497,-48.137,388.571,-77.991,87.486,-77.954
C01200=1012.496,-47.745,388.541,-77.749,87.479,-77.711
C01201=1012.496,-47.352,388.511,-77.535,87.472,-77.496
C01202=1012.497,-46.959,388.480,-77.329,87.465,-77.290
C01203=1012.497,-46.566,388.450,-77.135,87.459,-77.095
C01204=1012.496,-46.173,388.419,-76.951,87.454,-76.910
C01205=1012.496,-45.781,388.388,-76.775,87.448,-76.733
C01206=1012.496,-45.388,388.358,-76.619,87.443,-76.576
C01207=1012.496,-44.995,388.328,-76.471,87.438,-76.428
C01208=1012.496,-44.601,388.297,-76.333,87.433,-76.289
C01209=1012.495,-44.209,388.267,-76.212,87.429,-76.167
C01210=1012.496,-43.816,388.236,-76.101,87.426,-76.055
C01211=1012.495,-43.423,388.205,-76.006,87.423,-75.961
C01212=1012.496,-43.030,388.175,-75.922,87.420,-75.875
C01213=1012.496,-42.637,388.145,-75.844,87.417,-75.798
C01214=1012.495,-42.243,388.114,-75.786,87.416,-75.738
C01215=1012.495,-41.850,388.084,-75.734,87.414,-75.687
C01216=1012.495,-41.457,388.053,-75.692,87.412,-75.644
C01217=1012.495,-41.063,388.023,-75.666,87.411,-75.618
C01218=1012.495,-40.670,387.992,-75.650,87.411,-75.602
C01219=1012.495,-40.277,387.962,-75.634,87.411,-75.585
C01220=1012.495,-39.884,387.931,-75.634,87.411,-75.585
C01221=1012.495,-39.491,387.901,-75.660,87.412,-75.611
C01222=1012.495,-39.096,387.870,-75.686,87.413,-75.636
C01223=1012.495,-38.703,387.839,-75.721,87.415,-75.671
C01224=1012.495,-38.310,387.809,-75.773,87.417,-75.723
C01225=1012.494,-37.917,387.778,-75.825,87.419,-75.774
C01226=1012.495,-37.524,387.748,-75.903,87.422,-75.852
C01227=1012.494,-37.130,387.717,-75.981,87.425,-75.930
C01228=1012.494,-36.737,387.687,-76.075,87.428,-76.024
C01229=1012.494,-36.343,387.656,-76.180,87.432,-76.129
C01230=1012.494,-35.949,387.626,-76.301,87.437,-76.250
C01231=1012.494,-35.556,387.596,-76.423,87.441,-76.372
C01232=1012.494,-35.162,387.565,-76.572,87.446,-76.521
C01233=1012.493,-34.769,387.534,-76.721,87.451,-76.670
C01234=1012.494,-34.375,387.504,-76.881,87.457,-76.830
C01235=1012.493,-33.982,387.473,-77.058,87.463,-77.007
C01236=1012.493,-33.589,387.443,-77.253,87.470,-77.203
C01237=1012.493,-33.194,387.413,-77.459,87.477,-77.409
C01238=1012.493,-32.801,387.382,-77.667,87.484,-77.616
C01239=1012.493,-32.407,387.351,-77.892,87.491,-77.842
C01240=1012.493,-32.014,387.321,-78.146,87.499,-78.097
C01241=1012.492,-31.621,387.290,-78.385,87.507,-78.336
C01242=1012.492,-31.227,387.260,-78.671,87.516,-78.622
C01243=1012.492,-30.833,387.230,-78.941,87.524,-78.893
C01244=1012.492,-30.440,387.199,-79.248,87.533,-79.201
C01245=1012.492,-30.046,387.168,-79.540,87.542,-79.493
C01246=1012.492,-29.653,387.138,-79.863,87.552,-79.816
C01247=1012.491,-29.260,387.107,-80.217,87.562,-80.171
C01248=1012.492,-28.866,387.077,-80.563,87.572,-80.517
C01249=1012.491,-28.472,387.047,-80.941,87.582,-80.896
C01250=1012.491,-28.079,387.017,-81.334,87.593,-81.290
C01251=1012.491,-27.686,386.986,-81.719,87.603,-81.676
C01252=1012.491,-27.292,386.955,-82.137,87.614,-82.095
C01253=1012.491,-26.899,386.925,-82.573,87.626,-82.530
C01254=1012.491,-26.505,386.894,-83.030,87.637,-82.988
C01255=1012.491,-26.112,386.864,-83.492,87.649,-83.451
C01256=1012.490,-25.719,386.833,-83.977,87.660,-83.937
C01257=1012.490,-25.326,386.803,-84.480,87.672,-84.441
C01258=1012.489,-24.931,386.773,-85.006,87.684,-84.969
C01259=1012.490,-24.538,386.742,-85.553,87.696,-85.516
C01260=1012.489,-24.145,386.712,-86.105,87.708,-86.069
C01261=1012.489,-23.752,386.681,-86.681,87.720,-86.646
C01262=1012.489,-23.359,386.651,-87.298,87.732,-87.264
C01263=1012.489,-22.965,386.620,-87.902,87.744,-87.869
C01264=1012.489,-22.572,386.590,-88.551,87.756,-88.520
C01265=1012.488,-22.179,386.559,-89.223,87.769,-89.193
C01266=1012.488,-21.785,386.529,-89.902,87.781,-89.873
C01267=1012.488,-21.392,386.498,-90.588,87.792,-90.560
C01268=1012.488,-20.999,386.468,-91.318,87.804,-91.291
C01269=1012.488,-20.606,386.438,-92.075,87.816,-92.050
C01270=1012.487,-20.209,386.407,-92.858,87.828,-92.834
C01271=1012.488,-19.858,386.380,-93.556,87.837,-93.534
C01272=1012.487,-19.652,386.364,-93.972,87.843,-93.951
C01273=1012.487,-19.422,386.346,-94.468,87.850,-94.447
C01274=1012.487,-19.166,386.326,-95.006,87.857,-94.987
C01275=1012.487,-18.892,386.305,-95.605,87.864,-95.587
C01276=1012.487,-18.612,386.283,-96.228,87.872,-96.211
C01277=1012.486,-18.340,386.262,-96.835,87.879,-96.819
C01278=1012.486,-18.087,386.243,-97.427,87.885,-97.413
C01279=1012.486,-17.860,386.225,-97.943,87.891,-97.928
C01280=1012.486,-17.657,386.210,-98.441,87.896,-98.428
C01281=1012.486,-17.271,386.180,-99.384,87.905,-99.372
C01282=1012.486,-16.876,386.149,-100.355,87.914,-100.346
C01283=1012.485,-16.477,386.118,-101.354,87.922,-101.347
C01284=1012.485,-16.082,386.087,-102.382,87.930,-102.376
C01285=1012.485,-15.685,386.057,-103.438,87.937,-103.434
C01286=1012.485,-15.294,386.027,-104.479,87.943,-104.477
C01287=1012.484,-14.910,385.997,-105.548,87.949,-105.548
C01288=1012.484,-14.533,385.967,-106.600,87.954,-106.603
C01289=1012.484,-14.159,385.939,-107.680,87.959,-107.684
C01290=1012.484,-13.781,385.910,-108.784,87.962,-108.790
C01291=1012.484,-13.395,385.880,-109.934,87.965,-109.943
C01292=1012.484,-12.996,385.849,-111.173,87.968,-111.184
C01293=1012.483,-12.587,385.817,-112.434,87.969,-112.448
C01294=1012.483,-12.173,385.785,-113.720,87.970,-113.735
C01295=1012.482,-11.759,385.753,-115.024,87.969,-115.043
C01296=1012.482,-11.343,385.722,-116.370,87.967,-116.391
C01297=1012.482,-10.925,385.689,-117.712,87.964,-117.736
C01298=1012.482,-10.506,385.656,-119.068,87.960,-119.095
C01299=1012.481,-10.086,385.624,-120.466,87.954,-120.495
C01300=1012.482,-9.664,385.591,-121.848,87.948,-121.881
C01301=1012.481,-9.242,385.559,-123.246,87.940,-123.281
C01302=1012.481,-9.032,385.542,-123.948,87.935,-123.985
C01303=1012.481,-8.821,385.526,-124.673,87.930,-124.711
C01304=1012.481,-8.609,385.510,-125.385,87.925,-125.426
C01305=1012.481,-8.398,385.493,-126.102,87.919,-126.144
C01306=1012.481,-8.187,385.477,-126.790,87.913,-126.833
C01307=1012.481,-7.975,385.460,-127.515,87.907,-127.560
C01308=1012.480,-7.762,385.444,-128.235,87.900,-128.282
C01309=1012.481,-7.549,385.428,-128.951,87.893,-128.999
C01310=1012.480,-7.335,385.411,-129.661,87.885,-129.711
C01311=1012.480,-7.121,385.395,-130.366,87.877,-130.417
C01312=1012.480,-6.906,385.378,-131.105,87.869,-131.158
C01313=1012.480,-6.690,385.361,-131.799,87.860,-131.854
C01314=1012.479,-6.474,385.344,-132.526,87.851,-132.582
C01315=1012.479,-6.258,385.328,-133.246,87.841,-133.305
C01316=1012.479,-6.041,385.311,-133.960,87.831,-134.020
C01317=1012.479,-5.824,385.294,-134.681,87.821,-134.744
C01318=1012.479,-5.607,385.277,-135.381,87.810,-135.445
C01319=1012.479,-5.391,385.261,-136.074,87.799,-136.140
C01320=1012.478,-5.176,385.244,-136.773,87.787,-136.841
C01321=1012.478,-4.762,385.212,-138.123,87.764,-138.194
C01322=1012.479,-4.371,385.182,-139.360,87.741,-139.435
C01323=1012.478,-3.992,385.153,-140.547,87.717,-140.626
C01324=1012.478,-3.607,385.123,-141.744,87.691,-141.826
C01325=1012.478,-3.204,385.091,-142.979,87.664,-143.065
C01326=1012.477,-2.793,385.060,-144.228,87.633,-144.318
C01327=1012.476,-2.383,385.028,-145.465,87.602,-145.559
C01328=1012.477,-1.974,384.996,-146.648,87.569,-146.746
C01329=1012.476,-1.568,384.965,-147.819,87.535,-147.921
C01330=1012.477,-1.163,384.934,-148.966,87.500,-149.072
C01331=1012.476,-0.761,384.903,-150.072,87.464,-150.182
C01332=1012.476,-0.360,384.871,-151.153,87.427,-151.268
C01333=1012.476,0.038,384.841,-152.203,87.389,-152.322
C01334=1012.475,0.433,384.810,-153.241,87.350,-153.364
C01335=1012.475,0.827,384.780,-154.228,87.310,-154.356
C01336=1012.474,1.224,384.749,-155.210,87.268,-155.343
C01337=1012.474,1.621,384.718,-156.186,87.225,-156.323
C01338=1012.474,2.013,384.688,-157.108,87.182,-157.249
C01339=1012.474,2.384,384.659,-157.973,87.139,-158.119
C01340=1012.474,2.727,384.633,-158.746,87.100,-158.897
C01341=1012.474,3.050,384.608,-159.472,87.061,-159.626
C01342=1012.473,3.374,384.582,-160.183,87.022,-160.342
C01343=1012.473,3.717,384.556,-160.916,86.979,-161.078
C01344=1012.473,4.090,384.527,-161.686,86.933,-161.853
C01345=1012.473,4.481,384.497,-162.478,86.883,-162.651
C01346=1012.472,4.871,384.467,-163.260,86.832,-163.437
C01347=1012.472,5.260,384.437,-164.001,86.781,-164.184
C01348=1012.472,5.650,384.407,-164.747,86.728,-164.934
C01349=1012.472,6.043,384.377,-165.456,86.675,-165.650
C01350=1012.471,6.436,384.346,-166.173,86.619,-166.372
C01351=1012.472,6.826,384.315,-166.852,86.563,-167.056
C01352=1012.472,7.213,384.285,-167.506,86.508,-167.716
C01353=1012.471,7.594,384.257,-168.140,86.452,-168.355
C01354=1012.471,7.973,384.227,-168.753,86.396,-168.973
C01355=1012.471,8.348,384.198,-169.334,86.339,-169.560
C01356=1012.471,8.723,384.168,-169.908,86.282,-170.141
C01357=1012.470,9.096,384.140,-170.478,86.224,-170.716
C01358=1012.471,9.470,384.111,-171.018,86.165,-171.262
C01359=1012.470,9.845,384.082,-171.552,86.106,-171.802
C01360=1012.470,10.221,384.053,-172.071,86.045,-172.327
C01361=1012.470,10.599,384.024,-172.584,85.984,-172.846
C01362=1012.469,10.972,383.995,-173.081,85.923,-173.349
C01363=1012.469,11.337,383.967,-173.551,85.862,-173.825
C01364=1012.469,11.701,383.939,-174.008,85.800,-174.288
C01365=1012.469,12.074,383.910,-174.461,85.737,-174.748
C01366=1012.469,12.456,383.880,-174.920,85.672,-175.213
C01367=1012.468,12.840,383.850,-175.375,85.605,-175.674
C01368=1012.468,13.224,383.820,-175.805,85.538,-176.112
C01369=1012.468,13.606,383.791,-176.232,85.471,-176.544
C01370=1012.467,13.988,383.762,-176.645,85.402,-176.964
C01371=1012.467,14.369,383.732,-177.045,85.334,-177.372
C01372=1012.468,14.749,383.702,-177.441,85.264,-177.775
C01373=1012.467,15.130,383.673,-177.817,85.195,-178.159
C01374=1012.467,15.509,383.643,-178.190,85.124,-178.538
C01375=1012.467,15.891,383.614,-178.559,85.053,-178.914
C01376=1012.466,16.272,383.585,-178.917,84.981,-179.280
C01377=1012.467,16.655,383.555,-179.264,84.908,-179.634
C01378=1012.467,17.039,383.525,-179.607,84.834,-179.985
C01379=1012.466,17.425,383.495,-179.940,84.760,179.674
C01380=1012.467,17.813,383.465,179.730,84.684,179.337
C01381=1012.466,18.203,383.435,179.411,84.608,179.009
C01382=1012.466,18.595,383.404,179.095,84.530,178.685
C01383=1012.466,18.995,383.373,178.775,84.451,178.358
C01384=1012.466,19.398,383.343,178.467,84.370,178.040
C01385=1012.466,19.600,383.327,178.313,84.329,177.882
C01386=1012.466,19.822,383.310,178.152,84.284,177.715
C01387=1012.465,20.064,383.290,177.975,84.235,177.534
C01388=1012.466,20.324,383.270,177.787,84.182,177.340
C01389=1012.465,20.594,383.249,177.590,84.126,177.138
C01390=1012.465,20.862,383.229,177.404,84.070,176.946
C01391=1012.465,21.122,383.209,177.227,84.017,176.762
C01392=1012.465,21.371,383.190,177.057,83.965,176.587
C01393=1012.466,21.599,383.172,176.905,83.917,176.430
C01394=1012.465,21.987,383.141,176.653,83.836,176.168
C01395=1012.465,22.315,383.116,176.438,83.766,175.946
C01396=1012.464,22.647,383.091,176.230,83.695,175.730
C01397=1012.465,22.923,383.069,176.061,83.637,175.555
C01398=1012.465,23.288,383.040,175.840,83.558,175.325
C01399=1012.465,23.703,383.009,175.592,83.467,175.067
C01400=1012.464,24.044,382.982,175.395,83.394,174.862
C01401=1012.464,24.423,382.953,175.180,83.311,174.637
C01402=1012.465,24.819,382.922,174.959,83.223,174.406
C01403=1012.465,25.214,382.891,174.743,83.136,174.181
C01404=1012.464,25.611,382.860,174.535,83.048,173.963
C01405=1012.464,26.009,382.829,174.330,82.958,173.747
C01406=1012.464,26.407,382.799,174.124,82.868,173.531
C01407=1012.464,26.803,382.767,173.930,82.779,173.326
C01408=1012.465,27.198,382.737,173.741,82.689,173.127
C01409=1012.464,27.591,382.707,173.552,82.599,172.928
C01410=1012.464,27.985,382.676,173.369,82.508,172.735
C01411=1012.464,28.378,382.646,173.193,82.417,172.547
C01412=1012.464,28.771,382.615,173.017,82.325,172.360
C01413=1012.464,29.167,382.584,172.846,82.233,172.178
C01414=1012.464,29.561,382.554,172.681,82.140,172.002
C01415=1012.464,29.957,382.523,172.515,82.047,171.825
C01416=1012.464,30.352,382.492,172.356,81.953,171.654
C01417=1012.464,30.747,382.462,172.197,81.858,171.484
C01418=1012.464,31.143,382.431,172.042,81.763,171.318
C01419=1012.465,31.539,382.401,171.893,81.668,171.156
C01420=1012.463,31.934,382.370,171.747,81.573,170.998
C01421=1012.464,32.329,382.339,171.602,81.476,170.842
C01422=1012.464,32.725,382.308,171.462,81.380,170.689
C01423=1012.464,33.120,382.277,171.321,81.282,170.537
C01424=1012.464,33.515,382.247,171.188,81.186,170.392
C01425=1012.464,33.911,382.216,171.057,81.088,170.248
C01426=1012.465,34.306,382.185,170.925,80.989,170.104
C01427=1012.465,34.702,382.154,170.799,80.890,169.964
C01428=1012.465,35.097,382.123,170.674,80.791,169.827
C01429=1012.465,35.492,382.093,170.554,80.691,169.694
C01430=1012.465,35.888,382.062,170.434,80.591,169.561
C01431=1012.465,36.284,382.032,170.318,80.490,169.432
C01432=1012.465,36.679,382.000,170.205,80.390,169.305
C01433=1012.465,37.075,381.969,170.092,80.289,169.179
C01434=1012.466,37.470,381.938,169.984,80.186,169.057
C01435=1012.465,37.865,381.908,169.874,80.084,168.934
C01436=1012.466,38.261,381.877,169.772,79.982,168.817
C01437=1012.466,38.656,381.846,169.669,79.879,168.700
C01438=1012.466,39.052,381.815,169.566,79.775,168.584
C01439=1012.467,39.447,381.785,169.467,79.671,168.471
C01440=1012.467,39.843,381.754,169.371,79.567,168.360
C01441=1012.467,40.239,381.724,169.277,79.463,168.252
C01442=1012.467,40.634,381.693,169.183,79.358,168.144
C01443=1012.467,41.030,381.661,169.093,79.252,168.038
C01444=1012.467,41.426,381.630,169.003,79.146,167.933
C01445=1012.467,41.821,381.600,168.915,79.039,167.831
C01446=1012.468,42.217,381.569,168.829,78.933,167.730
C01447=1012.468,42.612,381.538,168.745,78.826,167.630
C01448=1012.468,43.008,381.507,168.662,78.718,167.533
C01449=1012.469,43.403,381.476,168.582,78.610,167.437
C01450=1012.469,43.800,381.446,168.506,78.502,167.344
C01451=1012.470,44.196,381.415,168.429,78.393,167.251
C01452=1012.470,44.591,381.384,168.351,78.284,167.158
C01453=1012.470,44.987,381.353,168.279,78.175,167.069
C01454=1012.470,45.382,381.322,168.203,78.065,166.978
C01455=1012.470,45.778,381.291,168.133,77.955,166.892
C01456=1012.471,46.174,381.260,168.063,77.844,166.805
C01457=1012.471,46.570,381.229,167.996,77.732,166.721
C01458=1012.472,46.965,381.198,167.927,77.621,166.636
C01459=1012.472,47.361,381.168,167.862,77.509,166.554
C01460=1012.472,47.757,381.136,167.798,77.397,166.473
C01461=1012.473,48.153,381.106,167.736,77.285,166.394
C01462=1012.473,48.548,381.075,167.675,77.172,166.315
C01463=1012.474,48.945,381.044,167.614,77.058,166.236
C01464=1012.474,49.340,381.013,167.554,76.944,166.159
C01465=1012.475,49.736,380.982,167.496,76.830,166.083
C01466=1012.475,50.133,380.951,167.439,76.715,166.008
C01467=1012.475,50.528,380.920,167.386,76.600,165.936
C01468=1012.476,50.925,380.889,167.330,76.484,165.863
C01469=1012.476,51.320,380.858,167.276,76.369,165.790
C01470=1012.477,51.716,380.827,167.224,76.252,165.720
C01471=1012.477,52.112,380.796,167.175,76.136,165.651
C01472=1012.478,52.508,380.764,167.124,76.019,165.582
C01473=1012.478,52.903,380.734,167.076,75.902,165.515
C01474=1012.479,53.300,380.703,167.028,75.784,165.448
C01475=1012.479,53.696,380.672,166.982,75.666,165.382
C01476=1012.480,54.092,380.641,166.935,75.547,165.316
C01477=1012.481,54.488,380.610,166.889,75.428,165.251
C01478=1012.481,54.884,380.578,166.847,75.309,165.188
C01479=1012.482,55.268,380.548,166.805,75.193,165.127
C01480=1012.482,55.676,380.516,166.762,75.069,165.063
C01481=1012.483,56.072,380.485,166.720,74.949,165.001
C01482=1012.484,56.469,380.455,166.680,74.828,164.941
C01483=1012.484,56.864,380.424,166.642,74.707,164.882
C01484=1012.485,57.261,380.392,166.603,74.585,164.822
C01485=1012.486,57.657,380.361,166.566,74.463,164.764
C01486=1012.486,58.052,380.330,166.530,74.341,164.706
C01487=1012.487,58.448,380.299,166.494,74.218,164.650
C01488=1012.488,58.845,380.268,166.459,74.094,164.593
C01489=1012.489,59.241,380.237,166.424,73.971,164.537
C01490=1012.489,59.636,380.206,166.393,73.847,164.483
C01491=1012.490,60.033,380.175,166.360,73.723,164.428
C01492=1012.491,60.429,380.143,166.328,73.598,164.374
C01493=1012.492,60.825,380.112,166.296,73.473,164.320
C01494=1012.493,61.221,380.081,166.267,73.347,164.268
C01495=1012.493,61.617,380.050,166.238,73.221,164.216
C01496=1012.494,62.013,380.019,166.209,73.095,164.165
C01497=1012.495,62.412,379.988,166.182,72.967,164.114
C01498=1012.495,62.696,379.966,166.162,72.876,164.078
C01499=1012.496,62.915,379.949,166.147,72.806,164.050
C01500=1012.497,63.157,379.930,166.131,72.728,164.019
C01501=1012.497,63.406,379.910,166.116,72.648,163.989
C01502=1012.497,63.640,379.892,166.099,72.571,163.959
C01503=1012.498,63.851,379.875,166.086,72.503,163.933
C01504=1012.498,64.257,379.838,166.081,72.469,163.921
C01505=1012.497,64.476,379.818,166.079,72.464,163.918
C01506=1012.497,64.702,379.797,166.079,72.459,163.917
C01507=1012.496,64.929,379.775,166.079,72.455,163.916
C01508=1012.496,65.152,379.755,166.079,72.451,163.915
C01509=1012.496,65.371,379.735,166.077,72.446,163.912
C01510=1012.494,65.586,379.714,166.077,72.441,163.911
C01511=1012.495,65.793,379.695,166.077,72.437,163.910
C01512=1012.493,66.187,379.658,166.075,72.429,163.907
C01513=1012.492,66.514,379.628,166.075,72.423,163.905
C01514=1012.492,66.877,379.594,166.074,72.414,163.902
C01515=1012.491,67.275,379.556,166.072,72.406,163.899
C01516=1012.491,67.673,379.519,166.072,72.397,163.896
C01517=1012.490,68.075,379.481,166.070,72.389,163.893
C01518=1012.489,68.486,379.443,166.070,72.380,163.891
C01519=1012.488,68.904,379.404,166.070,72.371,163.888
C01520=1012.486,69.320,379.364,166.068,72.362,163.885
C01521=1012.486,69.728,379.326,166.067,72.353,163.882
C01522=1012.484,70.132,379.288,166.066,72.345,163.879
C01523=1012.484,70.537,379.250,166.065,72.336,163.876
C01524=1012.483,70.942,379.212,166.065,72.328,163.873
C01525=1012.482,71.346,379.175,166.065,72.319,163.871
C01526=1012.481,71.750,379.137,166.063,72.309,163.867
C01527=1012.480,72.155,379.099,166.061,72.301,163.864
C01528=1012.479,72.562,379.060,166.061,72.292,163.862
C01529=1012.478,72.970,379.021,166.059,72.283,163.858
C01530=1012.477,73.379,378.982,166.059,72.274,163.856
C01531=1012.476,73.791,378.944,166.058,72.264,163.852
C01532=1012.476,74.206,378.905,166.057,72.255,163.850
C01533=1012.475,74.425,378.884,166.055,72.250,163.847
C01534=1012.474,74.653,378.862,166.056,72.246,163.846
C01535=1012.474,74.880,378.841,166.055,72.240,163.844
C01536=1012.473,75.095,378.821,166.055,72.235,163.843
C01537=1012.473,75.304,378.801,166.053,72.231,163.841
C01538=1012.471,75.718,378.761,166.054,72.221,163.839
C01539=1012.470,76.128,378.723,166.052,72.212,163.835
C01540=1012.469,76.529,378.685,166.051,72.203,163.832
C01541=1012.469,76.923,378.648,166.049,72.194,163.829
C01542=1012.468,77.310,378.611,166.049,72.185,163.826
C01543=1012.466,77.693,378.575,166.049,72.176,163.824
C01544=1012.466,78.073,378.539,166.048,72.168,163.821
C01545=1012.465,78.457,378.502,166.048,72.159,163.818
C01546=1012.464,78.846,378.465,166.046,72.149,163.815
C01547=1012.463,79.241,378.428,166.046,72.141,163.812
C01548=1012.462,79.643,378.390,166.044,72.131,163.809
C01549=1012.461,80.052,378.351,166.043,72.121,163.805
C01550=1012.460,80.464,378.312,166.041,72.112,163.802
C01551=1012.459,80.847,378.275,166.041,72.103,163.800
C01552=1012.458,81.211,378.240,166.041,72.094,163.797
C01553=1012.457,81.605,378.203,166.039,72.085,163.794
C01554=1012.456,82.019,378.164,166.039,72.076,163.791
C01555=1012.455,82.434,378.124,166.039,72.066,163.788
C01556=1012.454,82.846,378.085,166.037,72.056,163.785
C01557=1012.453,83.258,378.046,166.036,72.047,163.781
C01558=1012.452,83.669,378.006,166.035,72.036,163.778
C01559=1012.451,84.079,377.967,166.034,72.027,163.775
C01560=1012.450,84.487,377.928,166.034,72.017,163.772
C01561=1012.449,84.895,377.889,166.032,72.007,163.769
C01562=1012.447,85.300,377.850,166.032,71.997,163.766
C01563=1012.447,85.704,377.812,166.030,71.987,163.762
C01564=1012.446,86.107,377.773,166.030,71.977,163.760
C01565=1012.444,86.509,377.735,166.028,71.968,163.756
C01566=1012.443,86.910,377.697,166.028,71.957,163.753
C01567=1012.443,87.310,377.658,166.027,71.948,163.750
C01568=1012.441,87.703,377.620,166.026,71.938,163.747
C01569=1012.441,88.088,377.584,166.025,71.928,163.744
C01570=1012.440,88.466,377.547,166.025,71.919,163.741
C01571=1012.439,88.841,377.511,166.023,71.910,163.738
C01572=1012.438,89.219,377.474,166.022,71.900,163.734
C01573=1012.437,89.604,377.438,166.022,71.891,163.732
C01574=1012.435,90.000,377.399,166.022,71.881,163.729
C01575=1012.435,90.235,377.377,166.021,71.876,163.727
C01576=1012.434,90.509,377.350,166.020,71.869,163.725
C01577=1012.433,90.789,377.324,166.019,71.862,163.723
C01578=1012.433,91.035,377.300,166.019,71.856,163.721
C01579=1012.432,91.438,377.261,166.018,71.846,163.718
C01580=1012.430,91.832,377.224,166.018,71.836,163.715
C01581=1012.429,92.227,377.185,166.016,71.825,163.711
C01582=1012.429,92.622,377.147,166.014,71.814,163.707
C01583=1012.428,93.017,377.109,166.014,71.804,163.705
C01584=1012.426,93.411,377.071,166.014,71.794,163.702
C01585=1012.425,93.805,377.033,166.012,71.784,163.698
C01586=1012.425,94.201,376.995,166.013,71.776,163.696
C01587=1012.423,94.595,376.957,166.011,71.766,163.693
C01588=1012.422,94.989,376.919,166.011,71.756,163.690
C01589=1012.421,95.384,376.881,166.011,71.746,163.687
C01590=1012.421,95.779,376.842,166.009,71.735,163.683
C01591=1012.420,96.173,376.804,166.008,71.724,163.680
C01592=1012.418,96.568,376.766,166.007,71.712,163.676
C01593=1012.417,96.962,376.727,166.007,71.702,163.674
C01594=1012.415,97.357,376.689,166.006,71.693,163.670
C01595=1012.415,97.752,376.651,166.006,71.683,163.667
C01596=1012.414,98.146,376.613,166.004,71.673,163.664
C01597=1012.413,98.540,376.574,166.004,71.663,163.661
C01598=1012.412,98.935,376.537,166.003,71.652,163.658
C01599=1012.411,99.329,376.498,166.002,71.640,163.654
C01600=1012.409,99.724,376.460,166.002,71.629,163.651
C01601=1012.408,100.119,376.421,166.001,71.618,163.648
C01602=1012.407,100.513,376.383,166.001,71.608,163.645
C01603=1012.406,100.907,376.345,165.999,71.598,163.642
C01604=1012.405,101.301,376.306,165.999,71.588,163.639
C01605=1012.403,101.696,376.268,165.999,71.578,163.636
C01606=1012.402,102.090,376.229,165.998,71.567,163.632
C01607=1012.402,102.485,376.190,165.997,71.556,163.629
C01608=1012.401,102.880,376.153,165.997,71.544,163.626
C01609=1012.400,103.274,376.114,165.996,71.532,163.622
C01610=1012.399,103.668,376.076,165.996,71.522,163.619
C01611=1012.397,104.063,376.037,165.994,71.512,163.616
C01612=1012.396,104.457,375.999,165.994,71.502,163.613
C01613=1012.395,104.851,375.960,165.993,71.491,163.610
C01614=1012.394,105.246,375.921,165.993,71.480,163.606
C01615=1012.393,105.640,375.882,165.991,71.469,163.603
C01616=1012.392,106.035,375.845,165.991,71.457,163.600
C01617=1012.391,106.429,375.806,165.991,71.444,163.596
C01618=1012.389,106.823,375.767,165.991,71.434,163.593
C01619=1012.388,107.217,375.729,165.991,71.424,163.591
C01620=1012.388,107.612,375.690,165.989,71.413,163.587
C01621=1012.386,108.006,375.651,165.988,71.402,163.583
C01622=1012.385,108.401,375.613,165.989,71.392,163.581
C01623=1012.384,108.795,375.574,165.986,71.380,163.577
C01624=1012.383,109.189,375.536,165.988,71.368,163.574
C01625=1012.381,109.583,375.497,165.986,71.356,163.570
C01626=1012.381,109.978,375.458,165.986,71.344,163.567
C01627=1012.379,110.372,375.419,165.986,71.334,163.564
C01628=1012.378,110.766,375.380,165.985,71.323,163.561
C01629=1012.378,111.160,375.342,165.985,71.313,163.558
C01630=1012.376,111.555,375.303,165.985,71.302,163.555
C01631=1012.375,111.949,375.264,165.983,71.289,163.551
C01632=1012.375,112.343,375.225,165.983,71.278,163.548
C01633=1012.373,112.738,375.186,165.983,71.265,163.544
C01634=1012.372,113.132,375.148,165.981,71.253,163.540
C01635=1012.370,113.526,375.109,165.982,71.243,163.538
C01636=1012.369,113.920,375.070,165.981,71.231,163.535
C01637=1012.368,114.315,375.031,165.982,71.221,163.532
C01638=1012.367,114.709,374.992,165.980,71.209,163.528
C01639=1012.366,115.103,374.953,165.980,71.197,163.525
C01640=1012.365,115.497,374.914,165.980,71.186,163.522
C01641=1012.363,115.891,374.875,165.980,71.173,163.518
C01642=1012.363,116.286,374.836,165.979,71.161,163.515
C01643=1012.362,116.680,374.798,165.979,71.149,163.511
C01644=1012.360,117.075,374.759,165.979,71.138,163.508
C01645=1012.359,117.469,374.719,165.977,71.127,163.505
C01646=1012.359,117.863,374.680,165.977,71.116,163.502
C01647=1012.357,118.257,374.641,165.979,71.104,163.499
C01648=1012.356,118.651,374.602,165.977,71.091,163.495
C01649=1012.354,119.046,374.563,165.977,71.079,163.492
C01650=1012.354,119.440,374.524,165.976,71.066,163.488
C01651=1012.353,119.834,374.485,165.976,71.054,163.485
C01652=1012.352,120.228,374.446,165.976,71.043,163.482
C01653=1012.351,120.623,374.407,165.976,71.032,163.479
C01654=1012.349,121.018,374.368,165.975,71.020,163.475
C01655=1012.348,121.411,374.328,165.976,71.008,163.473
C01656=1012.347,121.805,374.289,165.975,70.995,163.469
C01657=1012.346,122.200,374.250,165.975,70.983,163.465
C01658=1012.345,122.594,374.211,165.975,70.970,163.462
C01659=1012.343,122.988,374.172,165.975,70.957,163.459
C01660=1012.342,123.383,374.132,165.975,70.946,163.456
C01661=1012.341,123.777,374.094,165.975,70.934,163.453
C01662=1012.340,124.171,374.054,165.975,70.923,163.450
C01663=1012.339,124.566,374.014,165.974,70.911,163.446
C01664=1012.338,124.960,373.976,165.974,70.898,163.443
C01665=1012.337,125.354,373.936,165.974,70.885,163.439
C01666=1012.335,125.749,373.897,165.974,70.872,163.436
C01667=1012.335,126.142,373.857,165.974,70.859,163.433
C01668=1012.334,126.537,373.818,165.974,70.847,163.429
C01669=1012.332,126.932,373.779,165.974,70.835,163.426
C01670=1012.331,127.326,373.739,165.974,70.824,163.423
C01671=1012.330,127.720,373.700,165.974,70.811,163.420
C01672=1012.329,128.114,373.660,165.973,70.799,163.416
C01673=1012.328,128.509,373.621,165.973,70.786,163.413
C01674=1012.326,128.903,373.582,165.974,70.773,163.410
C01675=1012.325,129.298,373.542,165.973,70.759,163.406
C01676=1012.324,129.692,373.503,165.973,70.746,163.403
C01677=1012.323,130.086,373.462,165.973,70.735,163.400
C01678=1012.322,130.480,373.424,165.975,70.723,163.397
C01679=1012.321,130.875,373.384,165.974,70.711,163.394
C01680=1012.320,131.270,373.344,165.974,70.698,163.390
C01681=1012.319,131.664,373.305,165.975,70.684,163.387
C01682=1012.318,132.059,373.265,165.974,70.671,163.383
C01683=1012.316,132.452,373.225,165.974,70.658,163.380
C01684=1012.315,132.847,373.186,165.974,70.644,163.376
C01685=1012.314,133.241,373.146,165.974,70.633,163.374
C01686=1012.313,133.636,373.107,165.975,70.620,163.370
C01687=1012.312,134.031,373.066,165.975,70.607,163.367
C01688=1012.310,134.425,373.027,165.975,70.594,163.364
C01689=1012.310,134.819,372.987,165.975,70.582,163.361
C01690=1012.309,135.050,372.965,165.977,70.574,163.359
C01691=1012.308,135.310,372.938,165.976,70.564,163.357
C01692=1012.307,135.720,372.897,165.976,70.550,163.353
C01693=1012.306,136.088,372.860,165.976,70.537,163.350
C01694=1012.305,136.430,372.825,165.977,70.526,163.347
C01695=1012.305,136.750,372.793,165.977,70.516,163.345
C01696=1012.304,137.072,372.761,165.976,70.505,163.341
C01697=1012.303,137.415,372.726,165.977,70.494,163.338
C01698=1012.301,137.763,372.691,165.978,70.482,163.336
C01699=1012.301,138.064,372.661,165.979,70.472,163.334
C01700=1012.300,138.460,372.620,165.979,70.459,163.331
C01701=1012.299,138.680,372.598,165.978,70.451,163.328
C01702=1012.299,138.915,372.574,165.979,70.443,163.327
C01703=1012.297,139.163,372.549,165.980,70.435,163.325
C01704=1012.297,139.421,372.524,165.980,70.426,163.323
C01705=1012.296,139.684,372.497,165.980,70.418,163.320
C01706=1012.295,139.945,372.471,165.979,70.409,163.317
C01707=1012.295,140.199,372.445,165.979,70.400,163.315
C01708=1012.294,140.441,372.420,165.981,70.392,163.314
C01709=1012.293,140.668,372.398,165.981,70.384,163.312
C01710=1012.293,140.879,372.376,165.980,70.377,163.310
C01711=1012.293,141.097,372.354,165.981,70.370,163.308
C01712=1012.291,141.502,372.312,165.981,70.356,163.305
C01713=1012.290,141.767,372.286,165.982,70.347,163.303
C01714=1012.290,141.967,372.266,165.983,70.340,163.301
C01715=1012.289,142.368,372.224,165.984,70.326,163.299
C01716=1012.288,142.770,372.184,165.984,70.312,163.295
C01717=1012.286,143.171,372.143,165.983,70.299,163.291
C01718=1012.286,143.574,372.103,165.985,70.285,163.288
C01719=1012.284,143.978,372.061,165.985,70.271,163.285
C01720=1012.284,144.381,372.020,165.985,70.257,163.281
C01721=1012.283,144.786,371.979,165.987,70.243,163.278
C01722=1012.282,145.191,371.938,165.988,70.229,163.276
C01723=1012.280,145.596,371.897,165.989,70.215,163.272
C01724=1012.279,146.002,371.856,165.989,70.201,163.269
C01725=1012.278,146.407,371.814,165.989,70.187,163.265
C01726=1012.277,146.814,371.773,165.991,70.172,163.262
C01727=1012.276,147.222,371.731,165.991,70.158,163.259
C01728=1012.164,147.180,371.322,168.817,78.669,167.619
C01729=1012.165,146.771,371.363,168.825,78.684,167.630
C01730=1012.166,146.365,371.404,168.834,78.698,167.641
C01731=1012.168,145.959,371.446,168.841,78.713,167.652
C01732=1012.168,145.553,371.487,168.850,78.727,167.664
C01733=1012.170,145.148,371.528,168.858,78.742,167.675
C01734=1012.171,144.743,371.569,168.867,78.756,167.687
C01735=1012.173,144.338,371.610,168.873,78.769,167.696
C01736=1012.173,143.935,371.651,168.881,78.784,167.707
C01737=1012.175,143.532,371.692,168.890,78.798,167.719
C01738=1012.175,143.129,371.733,168.899,78.813,167.731
C01739=1012.176,142.726,371.773,168.906,78.826,167.740
C01740=1012.178,142.325,371.814,168.915,78.840,167.752
C01741=1012.179,141.925,371.856,168.924,78.854,167.764
C01742=1012.180,141.725,371.875,168.927,78.861,167.769
C01743=1012.181,141.460,371.902,168.933,78.870,167.777
C01744=1012.182,141.054,371.943,168.943,78.884,167.789
C01745=1012.182,140.836,371.965,168.945,78.892,167.793
C01746=1012.183,140.625,371.987,168.951,78.899,167.800
C01747=1012.184,140.398,372.010,168.956,78.907,167.807
C01748=1012.184,140.156,372.034,168.960,78.916,167.813
C01749=1012.185,139.902,372.060,168.964,78.924,167.819
C01750=1012.186,139.641,372.086,168.971,78.933,167.827
C01751=1012.186,139.379,372.112,168.978,78.942,167.835
C01752=1012.188,139.121,372.139,168.982,78.951,167.841
C01753=1012.189,138.872,372.164,168.987,78.959,167.848
C01754=1012.189,138.637,372.188,168.991,78.967,167.854
C01755=1012.190,138.418,372.210,168.997,78.975,167.861
C01756=1012.190,138.021,372.249,169.008,78.988,167.874
C01757=1012.192,137.721,372.280,169.012,78.999,167.881
C01758=1012.193,137.372,372.315,169.019,79.010,167.890
C01759=1012.194,137.029,372.350,169.028,79.022,167.902
C01760=1012.195,136.708,372.383,169.032,79.033,167.909
C01761=1012.196,136.387,372.414,169.041,79.043,167.919
C01762=1012.197,136.047,372.449,169.048,79.055,167.928
C01763=1012.198,135.678,372.485,169.056,79.067,167.939
C01764=1012.199,135.267,372.527,169.067,79.083,167.953
C01765=1012.199,135.008,372.554,169.072,79.091,167.959
C01766=1012.200,134.777,372.576,169.077,79.099,167.966
C01767=1012.202,134.382,372.617,169.087,79.113,167.979
C01768=1012.203,133.988,372.656,169.096,79.126,167.990
C01769=1012.204,133.593,372.696,169.104,79.139,168.001
C01770=1012.206,133.199,372.735,169.113,79.151,168.012
C01771=1012.207,132.805,372.775,169.120,79.163,168.021
C01772=1012.208,132.410,372.814,169.130,79.177,168.034
C01773=1012.209,132.016,372.855,169.140,79.191,168.047
C01774=1012.210,131.622,372.893,169.148,79.204,168.057
C01775=1012.211,131.227,372.933,169.157,79.217,168.068
C01776=1012.212,130.833,372.972,169.168,79.231,168.082
C01777=1012.213,130.438,373.012,169.174,79.243,168.091
C01778=1012.215,130.044,373.052,169.184,79.255,168.103
C01779=1012.216,129.649,373.091,169.193,79.267,168.114
C01780=1012.217,129.256,373.131,169.202,79.280,168.125
C01781=1012.219,128.861,373.170,169.210,79.293,168.136
C01782=1012.220,128.466,373.209,169.222,79.307,168.150
C01783=1012.221,128.072,373.249,169.231,79.320,168.161
C01784=1012.222,127.678,373.288,169.240,79.332,168.173
C01785=1012.223,127.284,373.328,169.249,79.345,168.184
C01786=1012.225,126.890,373.367,169.259,79.357,168.196
C01787=1012.226,126.495,373.406,169.266,79.369,168.206
C01788=1012.227,126.101,373.446,169.276,79.381,168.218
C01789=1012.228,125.707,373.485,169.284,79.395,168.229
C01790=1012.229,125.312,373.524,169.296,79.408,168.243
C01791=1012.231,124.918,373.564,169.306,79.421,168.254
C01792=1012.232,124.524,373.603,169.315,79.434,168.266
C01793=1012.233,124.129,373.642,169.326,79.446,168.279
C01794=1012.234,123.735,373.682,169.332,79.458,168.288
C01795=1012.236,123.341,373.721,169.343,79.470,168.300
C01796=1012.237,122.947,373.760,169.351,79.481,168.311
C01797=1012.237,122.552,373.799,169.360,79.494,168.322
C01798=1012.239,122.158,373.839,169.370,79.506,168.334
C01799=1012.241,121.764,373.878,169.382,79.520,168.349
C01800=1012.242,121.370,373.916,169.389,79.532,168.358
C01801=1012.243,120.975,373.956,169.400,79.544,168.371
C01802=1012.244,120.581,373.995,169.411,79.556,168.384
C01803=1012.245,120.187,374.034,169.419,79.567,168.394
C01804=1012.247,119.793,374.073,169.427,79.579,168.404
C01805=1012.249,119.398,374.112,169.437,79.591,168.417
C01806=1012.249,119.004,374.152,169.447,79.604,168.429
C01807=1012.250,118.610,374.191,169.458,79.616,168.442
C01808=1012.251,118.216,374.229,169.468,79.629,168.454
C01809=1012.253,117.821,374.268,169.479,79.641,168.467
C01810=1012.255,117.427,374.307,169.488,79.652,168.477
